THIS^.AssertEquals_BOOL(
	Expected 	:= assertionIsWrong,
	Actual 		:= THIS^.assertorContainer.wasAssertionWrong,
	Message 	:= messageStringBuilder.sOut
);
END_METHOD

(*

short summary
==================
This test method tests ``assert.times.long.valueIsEqualTo``
method of CNM_AssertionInterfaces library, 
it provides the possibility to handover test data via parameter 


.. <legal notes>

legal notes
=================
| SPDX-FileCopyrightText: © 2022 ekvip automation GmbH <info@ekvip.de>
| SPDX-License-Identifier: Apache-2.0
| For details check: Apache-2.0_

.. _Apache-2.0: https://www.apache.org/licenses/LICENSE-2.0

.. </legal notes>

parameters
==========

*)

METHOD testValueIsEqualTo 
VAR_INPUT
	(* for the test it's the parameter ``currentValue`` *)
	valueToTest	:LTIME;
	(* for the test it's the parameter ``expectedValue`` *)
	expected	:LTIME;
END_VAR
VAR
	(* just the expectation if the assertion to test must be worng or true *)
	assertionIsWrong		:BOOL;
	(* contains the format string for the test message *)
	message					:Tc2_System.T_MaxString;
	(* TwinCAT printf with the test message *)
	messageStringBuilder	:Tc2_Utilities.FB_FormatString;
	(* LTIME value of ``currentValue`` as string *)
	currentValueAsString	:STRING(22);
	(* LTIME value of ``expectedValue`` as string *)
	expectedValueAsString	:STRING(22);
END_VAR
THIS^.assertorContainer.resetAssertor();

assertionIsWrong := (valueToTest <> expected);

message := SEL(
	assertionIsWrong,
	'currentValue is %s expectedValue is %s assertion must be TRUE', 
	'currentValue is %s expectedValue is %s assertion must be FALSE'
);
currentValueAsString := TO_STRING(valueToTest);
expectedValueAsString := TO_STRING(expected);

messageStringBuilder(
	sFormat := message,
	arg1 := THIS^.AnyToArg(currentValueAsString),
	arg2 := THIS^.AnyToArg(expectedValueAsString)
);

THIS^.assertorContainer.assertor.assert.times.long.valueIsEqualTo(
	currentValue	:= valueToTest,
	expectedValue	:= expected,
	message			:= ''
);

THIS^.AssertEquals_BOOL(
	Expected 	:= assertionIsWrong,
	Actual 		:= THIS^.assertorContainer.wasAssertionWrong,
	Message 	:= messageStringBuilder.sOut
);
END_METHOD

(*

short summary
==================
This test method tests ``assert.times.long.valueIsGreaterThan``
method of CNM_AssertionInterfaces library, 
it provides the possibility to handover test data via parameter 


.. <legal notes>

legal notes
=================
| SPDX-FileCopyrightText: © 2022 ekvip automation GmbH <info@ekvip.de>
| SPDX-License-Identifier: Apache-2.0
| For details check: Apache-2.0_

.. _Apache-2.0: https://www.apache.org/licenses/LICENSE-2.0

.. </legal notes>

parameters
==========

*)

METHOD testValueIsGreaterThan 
VAR_INPUT
	(* for the test it's the parameter ``currentValue`` *)
	valueToTest	:LTIME;
	(* for the test it's the parameter ``lessValue`` *)
	lessValue	:LTIME;
END_VAR
VAR
	(* just the expectation if the assertion to test must be worng or true *)
	assertionIsWrong		:BOOL;
	(* contains the format string for the test message *)
	message					:Tc2_System.T_MaxString;
	(* TwinCAT printf with the test message *)
	messageStringBuilder	:Tc2_Utilities.FB_FormatString;
	(* LTIME value of ``currentValue`` as string *)
	currentValueAsString	:STRING(22);
	(* LTIME value of ``lessValue`` as string *)
	lessValueAsString		:STRING(22);
END_VAR
THIS^.assertorContainer.resetAssertor();

assertionIsWrong := (valueToTest <= lessValue);

message := SEL(
	assertionIsWrong,
	'currentValue is %s lessValue is %s assertion must be TRUE', 
	'currentValue is %s lessValue is %s assertion must be FALSE'
);
currentValueAsString := TO_STRING(valueToTest);
lessValueAsString := TO_STRING(lessValue);

messageStringBuilder(
	sFormat := message,
	arg1 := THIS^.AnyToArg(currentValueAsString),
	arg2 := THIS^.AnyToArg(lessValueAsString)
);

THIS^.assertorContainer.assertor.assert.times.long.valueIsGreaterThan(
	currentValue	:= valueToTest,
	lessValue		:= lessValue,
	message			:= ''
);

THIS^.AssertEquals_BOOL(
	Expected 	:= assertionIsWrong,
	Actual 		:= THIS^.assertorContainer.wasAssertionWrong,
	Message 	:= messageStringBuilder.sOut
);
END_METHOD

(*

short summary
==================
This test method tests ``assert.times.long.valueIsInRangeOf``
method of CNM_AssertionInterfaces library, 
it provides the possibility to handover test data via parameter 


.. <legal notes>

legal notes
=================
| SPDX-FileCopyrightText: © 2022 ekvip automation GmbH <info@ekvip.de>
| SPDX-License-Identifier: Apache-2.0
| For details check: Apache-2.0_

.. _Apache-2.0: https://www.apache.org/licenses/LICENSE-2.0

.. </legal notes>

parameters
==========

*)

METHOD testValueIsInRangeOf 
VAR_INPUT
	(* for the test it's the parameter ``lowerLimit`` *)
	lowerLimit	:LTIME;
	(* for the test it's the parameter ``currentValue`` *)
	valueToTest	:LTIME;
	(* for the test it's the parameter ``upperLimit`` *)
	upperLimit	:LTIME;
END_VAR
VAR
	(* just the expectation if the assertion to test must be worng or true *)
	assertionIsWrong		:BOOL;
	(* contains the format string for the test message *)
	message					:Tc2_System.T_MaxString;
	(* TwinCAT printf with the test message *)
	messageStringBuilder	:Tc2_Utilities.FB_FormatString;
	(* LTIME value of ``lowerLimit`` as string *)
	lowerLimitAsString		:STRING(22);
	(* LTIME value of ``currentValue`` as string *)
	currentValueAsString	:STRING(22);
	(* LTIME value of ``upperLimit`` as string *)
	upperLimitAsString		:STRING(22);

END_VAR
THIS^.assertorContainer.resetAssertor();

assertionIsWrong := ((
		valueToTest < lowerLimit
	) OR (
		valueToTest > upperLimit
	)
);

message := SEL(
	assertionIsWrong,
	'lowerLimit is %s currentValue is %s upperLimit is %s assertion must be TRUE', 
	'lowerLimit is %s currentValue is %s upperLimit is %s assertion must be FALSE'
);
lowerLimitAsString		:= TO_STRING(lowerLimit);
currentValueAsString	:= TO_STRING(valueToTest);
upperLimitAsString		:= TO_STRING(upperLimit);

messageStringBuilder(
	sFormat := message,
	arg1 := THIS^.AnyToArg(lowerLimitAsString),
	arg2 := THIS^.AnyToArg(currentValueAsString),
	arg3 := THIS^.AnyToArg(upperLimitAsString)
);

THIS^.assertorContainer.assertor.assert.times.long.valueIsInRangeOf(
	lowerLimit		:= lowerLimit,
	currentValue	:= valueToTest,
	upperLimit		:= upperLimit,
	message			:= ''
);

THIS^.AssertEquals_BOOL(
	Expected 	:= assertionIsWrong,
	Actual 		:= THIS^.assertorContainer.wasAssertionWrong,
	Message 	:= messageStringBuilder.sOut
);
END_METHOD

(*

short summary
==================
This test method tests ``assert.times.long.valueIsLessThan``
method of CNM_AssertionInterfaces library, 
it provides the possibility to handover test data via parameter 


.. <legal notes>

legal notes
=================
| SPDX-FileCopyrightText: © 2022 ekvip automation GmbH <info@ekvip.de>
| SPDX-License-Identifier: Apache-2.0
| For details check: Apache-2.0_

.. _Apache-2.0: https://www.apache.org/licenses/LICENSE-2.0

.. </legal notes>

parameters
==========

*)

METHOD testValueIsLessThan 
VAR_INPUT
	(* for the test it's the parameter ``currentValue`` *)
	valueToTest		:LTIME;
	(* for the test it's the parameter ``greaterValue`` *)
	greaterValue	:LTIME;
END_VAR
VAR
	(* just the expectation if the assertion to test must be worng or true *)
	assertionIsWrong		:BOOL;
	(* contains the format string for the test message *)
	message					:Tc2_System.T_MaxString;
	(* TwinCAT printf with the test message *)
	messageStringBuilder	:Tc2_Utilities.FB_FormatString;
	(* LTIME value of ``currentValue`` as string *)
	currentValueAsString	:STRING(22);
	(* LTIME value of ``greaterValue`` as string *)
	greaterValueAsString	:STRING(22);
END_VAR
THIS^.assertorContainer.resetAssertor();

assertionIsWrong := (valueToTest >= greaterValue);

message := SEL(
	assertionIsWrong,
	'currentValue is %s greaterValue is %s assertion must be TRUE', 
	'currentValue is %s greaterValue is %s assertion must be FALSE'
);
currentValueAsString := TO_STRING(valueToTest);
greaterValueAsString := TO_STRING(greaterValue);

messageStringBuilder(
	sFormat := message,
	arg1 := THIS^.AnyToArg(currentValueAsString),
	arg2 := THIS^.AnyToArg(greaterValueAsString)
);

THIS^.assertorContainer.assertor.assert.times.long.valueIsLessThan(
	currentValue	:= valueToTest,
	greaterValue	:= greaterValue,
	message			:= ''
);

THIS^.AssertEquals_BOOL(
	Expected 	:= assertionIsWrong,
	Actual 		:= THIS^.assertorContainer.wasAssertionWrong,
	Message 	:= messageStringBuilder.sOut
);
END_METHOD

(*

short summary
==================
This test method tests ``assert.times.long.valueIsMax``
method of CNM_AssertionInterfaces library, 
it provides the possibility to handover test data via parameter 


.. <legal notes>

legal notes
=================
| SPDX-FileCopyrightText: © 2022 ekvip automation GmbH <info@ekvip.de>
| SPDX-License-Identifier: Apache-2.0
| For details check: Apache-2.0_

.. _Apache-2.0: https://www.apache.org/licenses/LICENSE-2.0

.. </legal notes>

parameters
==========

*)

METHOD testValueIsMax 
VAR_INPUT
	(* for the test it's the parameter ``currentValue`` *)
	valueToTest		:LTIME;
	(* for the test it's the parameter ``greaterValue`` *)
	maximumValue	:LTIME;
END_VAR
VAR
	(* just the expectation if the assertion to test must be worng or true *)
	assertionIsWrong		:BOOL;
	(* contains the format string for the test message *)
	message					:Tc2_System.T_MaxString;
	(* TwinCAT printf with the test message *)
	messageStringBuilder	:Tc2_Utilities.FB_FormatString;
	(* LTIME value of ``currentValue`` as string *)
	currentValueAsString	:STRING(22);
	(* LTIME value of ``maximumValue`` as string *)
	maximumValueAsString	:STRING(22);
END_VAR
THIS^.assertorContainer.resetAssertor();

assertionIsWrong := (valueToTest > maximumValue);

message := SEL(
	assertionIsWrong,
	'currentValue is %s maximumValue is %s assertion must be TRUE', 
	'currentValue is %s maximumValue is %s assertion must be FALSE'
);
currentValueAsString := TO_STRING(valueToTest);
maximumValueAsString := TO_STRING(maximumValue);

messageStringBuilder(
	sFormat := message,
	arg1 := THIS^.AnyToArg(currentValueAsString),
	arg2 := THIS^.AnyToArg(maximumValueAsString)
);

THIS^.assertorContainer.assertor.assert.times.long.valueIsMax(
	currentValue	:= valueToTest,
	maximumValue	:= maximumValue,
	message			:= ''
);

THIS^.AssertEquals_BOOL(
	Expected 	:= assertionIsWrong,
	Actual 		:= THIS^.assertorContainer.wasAssertionWrong,
	Message 	:= messageStringBuilder.sOut
);
END_METHOD

(*

short summary
==================
This test method tests ``assert.times.long.valueIsMin``
method of CNM_AssertionInterfaces library, 
it provides the possibility to handover test data via parameter 


.. <legal notes>

legal notes
=================
| SPDX-FileCopyrightText: © 2022 ekvip automation GmbH <info@ekvip.de>
| SPDX-License-Identifier: Apache-2.0
| For details check: Apache-2.0_

.. _Apache-2.0: https://www.apache.org/licenses/LICENSE-2.0

.. </legal notes>

parameters
==========

*)

METHOD testValueIsMin 
VAR_INPUT
	(* for the test it's the parameter ``currentValue`` *)
	valueToTest		:LTIME;
	(* for the test it's the parameter ``greaterValue`` *)
	minimumValue	:LTIME;
END_VAR
VAR
	(* just the expectation if the assertion to test must be worng or true *)
	assertionIsWrong		:BOOL;
	(* contains the format string for the test message *)
	message					:Tc2_System.T_MaxString;
	(* TwinCAT printf with the test message *)
	messageStringBuilder	:Tc2_Utilities.FB_FormatString;
	(* LTIME value of ``currentValue`` as string *)
	currentValueAsString	:STRING(22);
	(* LTIME value of ``minimumValue`` as string *)
	minimumValueAsString	:STRING(22);
END_VAR
THIS^.assertorContainer.resetAssertor();

assertionIsWrong := (valueToTest < minimumValue);

message := SEL(
	assertionIsWrong,
	'currentValue is %s minimumValue is %s assertion must be TRUE', 
	'currentValue is %s minimumValue is %s assertion must be FALSE'
);
currentValueAsString := TO_STRING(valueToTest);
minimumValueAsString := TO_STRING(minimumValue);

messageStringBuilder(
	sFormat := message,
	arg1 := THIS^.AnyToArg(currentValueAsString),
	arg2 := THIS^.AnyToArg(minimumValueAsString)
);

THIS^.assertorContainer.assertor.assert.times.long.valueIsMin(
	currentValue	:= valueToTest,
	minimumValue	:= minimumValue,
	message			:= ''
);

THIS^.AssertEquals_BOOL(
	Expected 	:= assertionIsWrong,
	Actual 		:= THIS^.assertorContainer.wasAssertionWrong,
	Message 	:= messageStringBuilder.sOut
);
END_METHOD

(*

short summary
==================
This test method tests ``assert.times.long.valueIsNotEqualTo``
method of CNM_AssertionInterfaces library, 
it provides the possibility to handover test data via parameter 


.. <legal notes>

legal notes
=================
| SPDX-FileCopyrightText: © 2022 ekvip automation GmbH <info@ekvip.de>
| SPDX-License-Identifier: Apache-2.0
| For details check: Apache-2.0_

.. _Apache-2.0: https://www.apache.org/licenses/LICENSE-2.0

.. </legal notes>

parameters
==========

*)

METHOD testValueIsNotEqualTo 
VAR_INPUT
	(* for the test it's the parameter ``currentValue`` *)
	valueToTest		:LTIME;
	(* for the test it's the parameter ``unexpectedValue`` *)
	unexpectedValue	:LTIME;
END_VAR
VAR
	(* just the expectation if the assertion to test must be worng or true *)
	assertionIsWrong		:BOOL;
	(* contains the format string for the test message *)
	message					:Tc2_System.T_MaxString;
	(* TwinCAT printf with the test message *)
	messageStringBuilder	:Tc2_Utilities.FB_FormatString;
	(* LTIME value of ``currentValue`` as string *)
	currentValueAsString	:STRING(22);
	(* LTIME value of ``unexpectedValue`` as string *)
	unexpectedValueAsString	:STRING(22);
END_VAR
THIS^.assertorContainer.resetAssertor();

assertionIsWrong := (valueToTest = unexpectedValue);

message := SEL(
	assertionIsWrong,
	'currentValue is %s expectedValue is %s assertion must be TRUE', 
	'currentValue is %s expectedValue is %s assertion must be FALSE'
);
currentValueAsString := TO_STRING(valueToTest);
unexpectedValueAsString := TO_STRING(unexpectedValue);

messageStringBuilder(
	sFormat := message,
	arg1 := THIS^.AnyToArg(currentValueAsString),
	arg2 := THIS^.AnyToArg(unexpectedValueAsString)
);

THIS^.assertorContainer.assertor.assert.times.long.valueIsNotEqualTo(
	currentValue	:= valueToTest,
	unexpectedValue	:= unexpectedValue,
	message			:= ''
);

THIS^.AssertEquals_BOOL(
	Expected 	:= assertionIsWrong,
	Actual 		:= THIS^.assertorContainer.wasAssertionWrong,
	Message 	:= messageStringBuilder.sOut
);
END_METHOD

END_FUNCTION_BLOCK

// ---- AssertionTester/AssertionTests/TimeAssertions/classes/TimeAssertionsTests.TcPOU
(*

short summary
==================
This class tests all methods of TIME assertions
with various combinations of inputs and checks expected 
outputs are satisfied or not

.. <legal notes>

legal notes
=================
| SPDX-FileCopyrightText: © 2022 ekvip automation GmbH <info@ekvip.de>
| SPDX-License-Identifier: Apache-2.0
| For details check: Apache-2.0_

.. _Apache-2.0: https://www.apache.org/licenses/LICENSE-2.0

.. </legal notes>

methods and properties
======================

*)


FUNCTION_BLOCK TimeAssertionsTests EXTENDS AbstractAssertorTest
VAR
	
END_VAR
VAR CONSTANT
	(* prefix to unify the test names *)
	TEST_NAME_PREFIX		:STRING := 'assert.times.simple.';
	(* max value of a DWORD *)
	{attribute 'hide'}
	MAX_DWORD				:DWORD := 16#FFFF_FFFF;
	(* min value of a DWORD *)
	{attribute 'hide'}
	MIN_DWORD				:DWORD := 16#0000_0000;
	(* only the msb is set *)
	{attribute 'hide'}
	MSB_ONLY				:DWORD := 16#8000_0000;
	(* only the msb is set *)
	{attribute 'hide'}
	LSB_ONLY				:DWORD := 16#0000_0001;
	(* all bits set except the msb *)
	{attribute 'hide'}
	WITHOUT_MSB 			:DWORD := 16#7FFF_FFFF;
	(* for every nibble is the msb set only *)
	{attribute 'hide'}
	ALL_NIBBLE_MSB			:DWORD := 16#8888_8888;
	(* for every nibble is the msb unset only *)
	{attribute 'hide'}
	WITHOUT_NIBBLE_MSB		:DWORD := 16#7777_7777;
	(* for every nibble is the lsb set only *)
	{attribute 'hide'}
	ALL_NIBBLE_LSB			:DWORD := 16#1111_1111;
	(* every bit is set except the lsb *)
	{attribute 'hide'}
	LSB_IS_UNSET			:DWORD := 16#FFFF_FFFE;
	(* max vale of time *)
	TIME_MAX				:TIME := TO_TIME(MAX_DWORD);
	(* min vale of time *)
	TIME_MIN				:TIME := TO_TIME(MIN_DWORD);
	(* only the msb is set *)
	TIME_MSB_ONLY			:TIME := TO_TIME(MSB_ONLY);
	(* all bits set except the msb *)
	TIME_WITHOUT_MSB 		:TIME := TO_TIME(WITHOUT_MSB);
	(* for every nibble is the msb set only *)
	TIME_ALL_NIBBLE_MSB		:TIME := TO_TIME(ALL_NIBBLE_MSB);
	(* for every nibble is the msb unset only *)
	TIME_WITHOUT_NIBBLE_MSB	:TIME := TO_TIME(WITHOUT_NIBBLE_MSB);
	(* for every nibble is the lsb set only *)
	TIME_ALL_NIBBLE_LSB		:TIME := TO_TIME(ALL_NIBBLE_LSB);	
	(* every bit is set except the lsb *)
	TIME_LSB_IS_UNSET		:TIME := TO_TIME(LSB_IS_UNSET);
	(* only the msb is set *)
	TIME_LSB_ONLY			:TIME := TO_TIME(LSB_ONLY);
END_VAR

THIS^.runTimeHasExpired();
THIS^.runTimeHasNotExpired();
THIS^.runValueIsEqualToTests();
THIS^.runValueIsGreaterThanTests();
THIS^.runValueIsInRangeOfTests();
THIS^.runValueIsLessThanTests();
THIS^.runValueIsMaxTests();
THIS^.runValueIsMinTests();
THIS^.runValueIsNotEqualToTests();

(*

short summary
==================
This test method is a helper function to create a unified test name

.. <legal notes>

legal notes
=================
| SPDX-FileCopyrightText: © 2022 ekvip automation GmbH <info@ekvip.de>
| SPDX-License-Identifier: Apache-2.0
| For details check: Apache-2.0_

.. _Apache-2.0: https://www.apache.org/licenses/LICENSE-2.0

.. </legal notes>

parameters
==========

*)

METHOD PROTECTED getTestNameFor :Tc2_System.T_MaxString
VAR_INPUT
	(* name of the method to test, to create a unified test name *)
	nameOfMethodToTest	:Tc2_System.T_MaxString;
END_VAR
getTestNameFor := Tc2_Standard.CONCAT(THIS^.TEST_NAME_PREFIX, nameOfMethodToTest);
END_METHOD

(*

short summary
=================
This method returns the passed time since the timestamp was created
(helper method of CNM_AssertionInterfaces)

.. <legal notes>

legal notes
=================
| SPDX-FileCopyrightText: © 2022 ekvip automation GmbH <info@ekvip.de>
| SPDX-License-Identifier: Apache-2.0
| For details check: Apache-2.0_

.. _Apache-2.0: https://www.apache.org/licenses/LICENSE-2.0

.. </legal notes>

parameters
=================
:return: passed time since ``startTime``

*)

METHOD PROTECTED getTimePassed :TIME
VAR_INPUT
	(* timestamp start *)
	startTime	:TIME;
END_VAR
VAR
	(* current time to calculate the passed time *)
	currentTime	:TIME;
END_VAR
currentTime := TIME();
IF (currentTime > startTime) THEN
	getTimePassed := (currentTime - startTime);
ELSE
	getTimePassed := ((THIS^.TIME_MAX - startTime) + currentTime);
END_IF
END_METHOD

(*

short summary
==================
This test method tests ``assert.times.simple.timeHasExpired``
method of CNM_AssertionInterfaces library with various inputs

.. <legal notes>

legal notes
=================
| SPDX-FileCopyrightText: © 2022 ekvip automation GmbH <info@ekvip.de>
| SPDX-License-Identifier: Apache-2.0
| For details check: Apache-2.0_

.. _Apache-2.0: https://www.apache.org/licenses/LICENSE-2.0

.. </legal notes>

*)

METHOD runTimeHasExpired
RETURN (NOT TcUnit.TEST_ORDERED(THIS^.getTestNameFor('timeHasExpired')));

THIS^.testTimeHasExpired(
	valueToTest := THIS^.TIME_MAX,
	expiring := THIS^.TIME_MAX
);
THIS^.testTimeHasExpired(
	valueToTest := THIS^.TIME_MIN,
	expiring := THIS^.TIME_MIN
);
THIS^.testTimeHasExpired(
	valueToTest := THIS^.TIME_MAX,
	expiring := THIS^.TIME_MIN
);
THIS^.testTimeHasExpired(
	valueToTest := THIS^.TIME_MIN,
	expiring := THIS^.TIME_MAX
);
THIS^.testTimeHasExpired(
	valueToTest := THIS^.TIME_ALL_NIBBLE_LSB,
	expiring := THIS^.TIME_ALL_NIBBLE_LSB
);	
THIS^.testTimeHasExpired(
	valueToTest := THIS^.TIME_ALL_NIBBLE_LSB,
	expiring := THIS^.TIME_ALL_NIBBLE_MSB
);
THIS^.testTimeHasExpired(
	valueToTest := THIS^.TIME_ALL_NIBBLE_MSB,
	expiring := THIS^.TIME_ALL_NIBBLE_LSB
);
THIS^.testTimeHasExpired(
	valueToTest := THIS^.TIME_LSB_ONLY,
	expiring := THIS^.TIME_MSB_ONLY
);
THIS^.testTimeHasExpired(
	valueToTest := THIS^.TIME_MSB_ONLY,
	expiring := THIS^.TIME_MSB_ONLY
);
THIS^.testTimeHasExpired(
	valueToTest := THIS^.TIME_MSB_ONLY,
	expiring := THIS^.TIME_LSB_ONLY
);
THIS^.testTimeHasExpired(
	valueToTest := THIS^.TIME_LSB_IS_UNSET,
	expiring := THIS^.TIME_MAX
);
THIS^.testTimeHasExpired(
	valueToTest := THIS^.TIME_MAX,
	expiring := THIS^.TIME_LSB_IS_UNSET
);

TcUnit.TEST_FINISHED();
END_METHOD

(*

short summary
==================
This test method tests ``assert.times.simple.timeHasNotExpired``
method of CNM_AssertionInterfaces library with various inputs

.. <legal notes>

legal notes
=================
| SPDX-FileCopyrightText: © 2022 ekvip automation GmbH <info@ekvip.de>
| SPDX-License-Identifier: Apache-2.0
| For details check: Apache-2.0_

.. _Apache-2.0: https://www.apache.org/licenses/LICENSE-2.0

.. </legal notes>

*)

METHOD runTimeHasNotExpired
RETURN (NOT TcUnit.TEST_ORDERED(THIS^.getTestNameFor('timeHasNotExpired')));

THIS^.testTimeHasExpired(
	valueToTest := THIS^.TIME_MAX,
	expiring := THIS^.TIME_MAX
);
THIS^.testTimeHasExpired(
	valueToTest := THIS^.TIME_MIN,
	expiring := THIS^.TIME_MIN
);
THIS^.testTimeHasExpired(
	valueToTest := THIS^.TIME_MAX,
	expiring := THIS^.TIME_MIN
);
THIS^.testTimeHasExpired(
	valueToTest := THIS^.TIME_MIN,
	expiring := THIS^.TIME_MAX
);
THIS^.testTimeHasExpired(
	valueToTest := THIS^.TIME_ALL_NIBBLE_LSB,
	expiring := THIS^.TIME_ALL_NIBBLE_LSB
);	
THIS^.testTimeHasExpired(
	valueToTest := THIS^.TIME_ALL_NIBBLE_LSB,
	expiring := THIS^.TIME_ALL_NIBBLE_MSB
);
THIS^.testTimeHasExpired(
	valueToTest := THIS^.TIME_ALL_NIBBLE_MSB,
	expiring := THIS^.TIME_ALL_NIBBLE_LSB
);
THIS^.testTimeHasExpired(
	valueToTest := THIS^.TIME_LSB_ONLY,
	expiring := THIS^.TIME_MSB_ONLY
);
THIS^.testTimeHasExpired(
	valueToTest := THIS^.TIME_MSB_ONLY,
	expiring := THIS^.TIME_MSB_ONLY
);
THIS^.testTimeHasExpired(
	valueToTest := THIS^.TIME_MSB_ONLY,
	expiring := THIS^.TIME_LSB_ONLY
);
THIS^.testTimeHasExpired(
	valueToTest := THIS^.TIME_LSB_IS_UNSET,
	expiring := THIS^.TIME_MAX
);
THIS^.testTimeHasExpired(
	valueToTest := THIS^.TIME_MAX,
	expiring := THIS^.TIME_LSB_IS_UNSET
);

TcUnit.TEST_FINISHED();
END_METHOD

(*

short summary
==================
This test method tests ``assert.times.simple.valueIsEqualTo``
method of CNM_AssertionInterfaces library with various inputs

.. <legal notes>

legal notes
=================
| SPDX-FileCopyrightText: © 2022 ekvip automation GmbH <info@ekvip.de>
| SPDX-License-Identifier: Apache-2.0
| For details check: Apache-2.0_

.. _Apache-2.0: https://www.apache.org/licenses/LICENSE-2.0

.. </legal notes>

*)

METHOD runValueIsEqualToTests
RETURN (NOT TcUnit.TEST_ORDERED(THIS^.getTestNameFor('valueIsEqualTo')));

THIS^.testValueIsEqualTo(
	valueToTest := THIS^.TIME_MAX,
	expected := THIS^.TIME_MAX
);
THIS^.testValueIsEqualTo(
	valueToTest := THIS^.TIME_MIN,
	expected := THIS^.TIME_MIN
);
THIS^.testValueIsEqualTo(
	valueToTest := THIS^.TIME_MIN,
	expected := THIS^.TIME_MAX
);
THIS^.testValueIsEqualTo(
	valueToTest := THIS^.TIME_MAX,
	expected := THIS^.TIME_MIN
);
THIS^.testValueIsEqualTo(
	valueToTest := THIS^.TIME_ALL_NIBBLE_LSB,
	expected := THIS^.TIME_ALL_NIBBLE_LSB
);
THIS^.testValueIsEqualTo(
	valueToTest := THIS^.TIME_LSB_ONLY,
	expected := THIS^.TIME_MSB_ONLY
);
THIS^.testValueIsEqualTo(
	valueToTest := THIS^.TIME_MSB_ONLY,
	expected := THIS^.TIME_MSB_ONLY
);
THIS^.testValueIsEqualTo(
	valueToTest := THIS^.TIME_MSB_ONLY,
	expected := THIS^.TIME_LSB_ONLY
);

TcUnit.TEST_FINISHED();
END_METHOD

(*

short summary
==================
This test method tests ``assert.times.simple.valueIsGreaterThan``
method of CNM_AssertionInterfaces library with various inputs

.. <legal notes>

legal notes
=================
| SPDX-FileCopyrightText: © 2022 ekvip automation GmbH <info@ekvip.de>
| SPDX-License-Identifier: Apache-2.0
| For details check: Apache-2.0_

.. _Apache-2.0: https://www.apache.org/licenses/LICENSE-2.0

.. </legal notes>

*)

METHOD runValueIsGreaterThanTests
RETURN (NOT TcUnit.TEST_ORDERED(THIS^.getTestNameFor('valueIsGreaterThan')));

THIS^.testValueIsGreaterThan(
	valueToTest := THIS^.TIME_MAX,
	lessValue := THIS^.TIME_MAX
);
THIS^.testValueIsGreaterThan(
	valueToTest := THIS^.TIME_MIN,
	lessValue := THIS^.TIME_MIN
);
THIS^.testValueIsGreaterThan(
	valueToTest := THIS^.TIME_MIN,
	lessValue := THIS^.TIME_MAX
);
THIS^.testValueIsGreaterThan(
	valueToTest := THIS^.TIME_MAX,
	lessValue := THIS^.TIME_MIN
);
THIS^.testValueIsGreaterThan(
	valueToTest := THIS^.TIME_ALL_NIBBLE_LSB,
	lessValue := THIS^.TIME_ALL_NIBBLE_LSB
);
THIS^.testValueIsGreaterThan(
	valueToTest := THIS^.TIME_ALL_NIBBLE_MSB,
	lessValue := THIS^.TIME_ALL_NIBBLE_LSB
);
THIS^.testValueIsGreaterThan(
	valueToTest := THIS^.TIME_ALL_NIBBLE_LSB,
	lessValue := THIS^.TIME_ALL_NIBBLE_MSB
);
THIS^.testValueIsGreaterThan(
	valueToTest := THIS^.TIME_LSB_ONLY,
	lessValue := THIS^.TIME_MSB_ONLY
);
THIS^.testValueIsGreaterThan(
	valueToTest := THIS^.TIME_MSB_ONLY,
	lessValue := THIS^.TIME_MSB_ONLY
);
THIS^.testValueIsGreaterThan(
	valueToTest := THIS^.TIME_MSB_ONLY,
	lessValue := THIS^.TIME_LSB_ONLY
);
THIS^.testValueIsGreaterThan(
	valueToTest := THIS^.TIME_LSB_IS_UNSET,
	lessValue := THIS^.TIME_MAX
);
THIS^.testValueIsGreaterThan(
	valueToTest := THIS^.TIME_MAX,
	lessValue := THIS^.TIME_LSB_IS_UNSET
);

TcUnit.TEST_FINISHED();
END_METHOD

(*

short summary
==================
This test method tests ``assert.times.simple.valueIsInRangeOf``
method of CNM_AssertionInterfaces library with various inputs

.. <legal notes>

legal notes
=================
| SPDX-FileCopyrightText: © 2022 ekvip automation GmbH <info@ekvip.de>
| SPDX-License-Identifier: Apache-2.0
| For details check: Apache-2.0_

.. _Apache-2.0: https://www.apache.org/licenses/LICENSE-2.0

.. </legal notes>

*)

METHOD runValueIsInRangeOfTests
RETURN (NOT TcUnit.TEST_ORDERED(THIS^.getTestNameFor('valueIsInRangeOf')));

THIS^.testValueIsInRangeOf(
	lowerLimit := THIS^.TIME_MIN,
	valueToTest := THIS^.TIME_MAX,
	upperLimit	:= THIS^.TIME_MAX
);
THIS^.testValueIsInRangeOf(
	lowerLimit := THIS^.TIME_MIN,
	valueToTest := THIS^.TIME_MIN,
	upperLimit	:= THIS^.TIME_MAX
);
THIS^.testValueIsInRangeOf(
	lowerLimit := THIS^.TIME_MAX,
	valueToTest := THIS^.TIME_MAX,
	upperLimit	:= THIS^.TIME_MIN
);
THIS^.testValueIsInRangeOf(
	lowerLimit := THIS^.TIME_MAX,
	valueToTest := THIS^.TIME_MIN,
	upperLimit	:= THIS^.TIME_MIN
);
THIS^.testValueIsInRangeOf(
	lowerLimit := THIS^.TIME_LSB_IS_UNSET,
	valueToTest := THIS^.TIME_MIN,
	upperLimit	:= THIS^.TIME_MAX
);
THIS^.testValueIsInRangeOf(
	lowerLimit := THIS^.TIME_MIN,
	valueToTest := THIS^.TIME_LSB_IS_UNSET,
	upperLimit	:= THIS^.TIME_MAX
);
THIS^.testValueIsInRangeOf(
	lowerLimit := THIS^.TIME_LSB_IS_UNSET,
	valueToTest := THIS^.TIME_LSB_IS_UNSET,
	upperLimit	:= THIS^.TIME_LSB_IS_UNSET
);
THIS^.testValueIsInRangeOf(
	lowerLimit := THIS^.TIME_ALL_NIBBLE_LSB,
	valueToTest := THIS^.TIME_LSB_IS_UNSET,
	upperLimit	:= THIS^.TIME_ALL_NIBBLE_MSB
);
THIS^.testValueIsInRangeOf(
	lowerLimit := THIS^.TIME_LSB_IS_UNSET,
	valueToTest := THIS^.TIME_ALL_NIBBLE_LSB,
	upperLimit	:= THIS^.TIME_ALL_NIBBLE_MSB
);
THIS^.testValueIsInRangeOf(
	lowerLimit := THIS^.TIME_LSB_ONLY,
	valueToTest := THIS^.TIME_WITHOUT_MSB,
	upperLimit	:= THIS^.TIME_MSB_ONLY
);
THIS^.testValueIsInRangeOf(
	lowerLimit := THIS^.TIME_WITHOUT_MSB,
	valueToTest := THIS^.TIME_LSB_ONLY,
	upperLimit	:= THIS^.TIME_MSB_ONLY
);
THIS^.testValueIsInRangeOf(
	lowerLimit := THIS^.TIME_WITHOUT_NIBBLE_MSB,
	valueToTest := THIS^.TIME_MAX,
	upperLimit	:= THIS^.TIME_ALL_NIBBLE_MSB
);
THIS^.testValueIsInRangeOf(
	lowerLimit := THIS^.TIME_WITHOUT_NIBBLE_MSB,
	valueToTest := THIS^.TIME_MIN,
	upperLimit	:= THIS^.TIME_ALL_NIBBLE_MSB
);
THIS^.testValueIsInRangeOf(
	lowerLimit := THIS^.TIME_WITHOUT_NIBBLE_MSB,
	valueToTest := THIS^.TIME_WITHOUT_NIBBLE_MSB,
	upperLimit	:= THIS^.TIME_ALL_NIBBLE_MSB
);
THIS^.testValueIsInRangeOf(
	lowerLimit := THIS^.TIME_WITHOUT_NIBBLE_MSB,
	valueToTest := THIS^.TIME_ALL_NIBBLE_MSB,
	upperLimit	:= THIS^.TIME_ALL_NIBBLE_MSB
);

TcUnit.TEST_FINISHED();
END_METHOD

(*

short summary
==================
This test method tests ``assert.times.simple.valueIsLessThan``
method of CNM_AssertionInterfaces library with various inputs

.. <legal notes>

legal notes
=================
| SPDX-FileCopyrightText: © 2022 ekvip automation GmbH <info@ekvip.de>
| SPDX-License-Identifier: Apache-2.0
| For details check: Apache-2.0_

.. _Apache-2.0: https://www.apache.org/licenses/LICENSE-2.0

.. </legal notes>

*)

METHOD runValueIsLessThanTests
RETURN (NOT TcUnit.TEST_ORDERED(THIS^.getTestNameFor('valueIsLessThan')));

THIS^.testValueIsLessThan(
	valueToTest := THIS^.TIME_MAX,
	greaterValue := THIS^.TIME_MAX
);
THIS^.testValueIsLessThan(
	valueToTest := THIS^.TIME_MIN,
	greaterValue := THIS^.TIME_MIN
);
THIS^.testValueIsLessThan(
	valueToTest := THIS^.TIME_MIN,
	greaterValue := THIS^.TIME_MAX
);
THIS^.testValueIsLessThan(
	valueToTest := THIS^.TIME_MAX,
	greaterValue := THIS^.TIME_MIN
);
THIS^.testValueIsLessThan(
	valueToTest := THIS^.TIME_ALL_NIBBLE_LSB,
	greaterValue := THIS^.TIME_ALL_NIBBLE_LSB
);
THIS^.testValueIsLessThan(
	valueToTest := THIS^.TIME_ALL_NIBBLE_MSB,
	greaterValue := THIS^.TIME_ALL_NIBBLE_LSB
);
THIS^.testValueIsLessThan(
	valueToTest := THIS^.TIME_ALL_NIBBLE_LSB,
	greaterValue := THIS^.TIME_ALL_NIBBLE_MSB
);
THIS^.testValueIsLessThan(
	valueToTest := THIS^.TIME_LSB_ONLY,
	greaterValue := THIS^.TIME_MSB_ONLY
);
THIS^.testValueIsLessThan(
	valueToTest := THIS^.TIME_MSB_ONLY,
	greaterValue := THIS^.TIME_MSB_ONLY
);
THIS^.testValueIsLessThan(
	valueToTest := THIS^.TIME_MSB_ONLY,
	greaterValue := THIS^.TIME_LSB_ONLY
);
THIS^.testValueIsLessThan(
	valueToTest := THIS^.TIME_LSB_IS_UNSET,
	greaterValue := THIS^.TIME_MAX
);
THIS^.testValueIsLessThan(
	valueToTest := THIS^.TIME_MAX,
	greaterValue := THIS^.TIME_LSB_IS_UNSET
);

TcUnit.TEST_FINISHED();
END_METHOD

(*

short summary
==================
This test method tests ``assert.times.simple.valueIsMax``
method of CNM_AssertionInterfaces library with various inputs

.. <legal notes>

legal notes
=================
| SPDX-FileCopyrightText: © 2022 ekvip automation GmbH <info@ekvip.de>
| SPDX-License-Identifier: Apache-2.0
| For details check: Apache-2.0_

.. _Apache-2.0: https://www.apache.org/licenses/LICENSE-2.0

.. </legal notes>

*)

METHOD runValueIsMaxTests
RETURN (NOT TcUnit.TEST_ORDERED(THIS^.getTestNameFor('valueIsMax')));

THIS^.testValueIsMax(
	valueToTest := THIS^.TIME_MAX,
	maximumValue := THIS^.TIME_MAX
);
THIS^.testValueIsMax(
	valueToTest := THIS^.TIME_MIN,
	maximumValue := THIS^.TIME_MIN
);
THIS^.testValueIsMax(
	valueToTest := THIS^.TIME_MIN,
	maximumValue := THIS^.TIME_MAX
);
THIS^.testValueIsMax(
	valueToTest := THIS^.TIME_MAX,
	maximumValue := THIS^.TIME_MIN
);
THIS^.testValueIsMax(
	valueToTest := THIS^.TIME_ALL_NIBBLE_LSB,
	maximumValue := THIS^.TIME_ALL_NIBBLE_LSB
);
THIS^.testValueIsMax(
	valueToTest := THIS^.TIME_ALL_NIBBLE_MSB,
	maximumValue := THIS^.TIME_ALL_NIBBLE_LSB
);
THIS^.testValueIsMax(
	valueToTest := THIS^.TIME_ALL_NIBBLE_LSB,
	maximumValue := THIS^.TIME_ALL_NIBBLE_MSB
);
THIS^.testValueIsMax(
	valueToTest := THIS^.TIME_LSB_ONLY,
	maximumValue := THIS^.TIME_MSB_ONLY
);
THIS^.testValueIsMax(
	valueToTest := THIS^.TIME_MSB_ONLY,
	maximumValue := THIS^.TIME_MSB_ONLY
);
THIS^.testValueIsMax(
	valueToTest := THIS^.TIME_MSB_ONLY,
	maximumValue := THIS^.TIME_LSB_ONLY
);
THIS^.testValueIsMax(
	valueToTest := THIS^.TIME_LSB_IS_UNSET,
	maximumValue := THIS^.TIME_MAX
);
THIS^.testValueIsMax(
	valueToTest := THIS^.TIME_MAX,
	maximumValue := THIS^.TIME_LSB_IS_UNSET
);

TcUnit.TEST_FINISHED();
END_METHOD

(*

short summary
==================
This test method tests ``assert.times.simple.valueIsMin``
method of CNM_AssertionInterfaces library with various inputs

.. <legal notes>

legal notes
=================
| SPDX-FileCopyrightText: © 2022 ekvip automation GmbH <info@ekvip.de>
| SPDX-License-Identifier: Apache-2.0
| For details check: Apache-2.0_

.. _Apache-2.0: https://www.apache.org/licenses/LICENSE-2.0

.. </legal notes>

*)

METHOD runValueIsMinTests
RETURN (NOT TcUnit.TEST_ORDERED(THIS^.getTestNameFor('valueIsMin')));

THIS^.testValueIsMin(
	valueToTest := THIS^.TIME_MAX,
	minimumValue := THIS^.TIME_MAX
);
THIS^.testValueIsMin(
	valueToTest := THIS^.TIME_MIN,
	minimumValue := THIS^.TIME_MIN
);
THIS^.testValueIsMin(
	valueToTest := THIS^.TIME_MIN,
	minimumValue := THIS^.TIME_MAX
);
THIS^.testValueIsMin(
	valueToTest := THIS^.TIME_MAX,
	minimumValue := THIS^.TIME_MIN
);
THIS^.testValueIsMin(
	valueToTest := THIS^.TIME_ALL_NIBBLE_LSB,
	minimumValue := THIS^.TIME_ALL_NIBBLE_LSB
);
THIS^.testValueIsMin(
	valueToTest := THIS^.TIME_ALL_NIBBLE_MSB,
	minimumValue := THIS^.TIME_ALL_NIBBLE_LSB
);
THIS^.testValueIsMin(
	valueToTest := THIS^.TIME_ALL_NIBBLE_LSB,
	minimumValue := THIS^.TIME_ALL_NIBBLE_MSB
);
THIS^.testValueIsMin(
	valueToTest := THIS^.TIME_LSB_ONLY,
	minimumValue := THIS^.TIME_MSB_ONLY
);
THIS^.testValueIsMin(
	valueToTest := THIS^.TIME_MSB_ONLY,
	minimumValue := THIS^.TIME_MSB_ONLY
);
THIS^.testValueIsMin(
	valueToTest := THIS^.TIME_MSB_ONLY,
	minimumValue := THIS^.TIME_LSB_ONLY
);
THIS^.testValueIsMin(
	valueToTest := THIS^.TIME_LSB_IS_UNSET,
	minimumValue := THIS^.TIME_MAX
);
THIS^.testValueIsMin(
	valueToTest := THIS^.TIME_MAX,
	minimumValue := THIS^.TIME_LSB_IS_UNSET
);

TcUnit.TEST_FINISHED();
END_METHOD

(*

short summary
==================
This test method tests ``assert.times.simple.valueIsNotEqualTo``
method of CNM_AssertionInterfaces library with various inputs

.. <legal notes>

legal notes
=================
| SPDX-FileCopyrightText: © 2022 ekvip automation GmbH <info@ekvip.de>
| SPDX-License-Identifier: Apache-2.0
| For details check: Apache-2.0_

.. _Apache-2.0: https://www.apache.org/licenses/LICENSE-2.0

.. </legal notes>

*)

METHOD runValueIsNotEqualToTests
RETURN (NOT TcUnit.TEST_ORDERED(THIS^.getTestNameFor('valueIsNotEqualTo')));

THIS^.testValueIsNotEqualTo(
	valueToTest := THIS^.TIME_MAX,
	unexpectedValue := THIS^.TIME_MAX
);
THIS^.testValueIsNotEqualTo(
	valueToTest := THIS^.TIME_MIN,
	unexpectedValue := THIS^.TIME_MIN
);
THIS^.testValueIsNotEqualTo(
	valueToTest := THIS^.TIME_MIN,
	unexpectedValue := THIS^.TIME_MAX
);
THIS^.testValueIsNotEqualTo(
	valueToTest := THIS^.TIME_MAX,
	unexpectedValue := THIS^.TIME_MIN
);
THIS^.testValueIsNotEqualTo(
	valueToTest := THIS^.TIME_ALL_NIBBLE_LSB,
	unexpectedValue := THIS^.TIME_ALL_NIBBLE_LSB
);
THIS^.testValueIsNotEqualTo(
	valueToTest := THIS^.TIME_LSB_ONLY,
	unexpectedValue := THIS^.TIME_MSB_ONLY
);
THIS^.testValueIsNotEqualTo(
	valueToTest := THIS^.TIME_MSB_ONLY,
	unexpectedValue := THIS^.TIME_MSB_ONLY
);
THIS^.testValueIsNotEqualTo(
	valueToTest := THIS^.TIME_MSB_ONLY,
	unexpectedValue := THIS^.TIME_LSB_ONLY
);

TcUnit.TEST_FINISHED();
END_METHOD

(*

short summary
==================
This test method tests ``assert.times.simple.timeHasExpired``
method of CNM_AssertionInterfaces library, 
it provides the possibility to handover test data via parameter 


.. <legal notes>

legal notes
=================
| SPDX-FileCopyrightText: © 2022 ekvip automation GmbH <info@ekvip.de>
| SPDX-License-Identifier: Apache-2.0
| For details check: Apache-2.0_

.. _Apache-2.0: https://www.apache.org/licenses/LICENSE-2.0

.. </legal notes>

parameters
==========

*)


METHOD testTimeHasExpired 
VAR_INPUT
	(* for the test it's the parameter ``timestamp`` *)
	valueToTest	:TIME;
	(* for the test it's the parameter ``expiringTime`` *)
	expiring	:TIME;
END_VAR
VAR
	(* just the expectation if the assertion to test must be wrong or true *)
	assertionIsWrong		:BOOL;
	(* contains the format string for the test message *)
	message					:Tc2_System.T_MaxString;
	(* TwinCAT printf with the test message *)
	messageStringBuilder	:Tc2_Utilities.FB_FormatString;
	(* TIME value of ``expiringTime`` as string *)
	expiringTimeAsString	:STRING(22);
	(* TIME value of ``expectedValue`` as string *)
	timestampAsString		:STRING(22);
END_VAR
THIS^.assertorContainer.resetAssertor();

assertionIsWrong := (getTimePassed(startTime := valueToTest) < expiring);

message := SEL(
	assertionIsWrong,
	'timestamp is %s expiringTime is %s assertion must be TRUE', 
	'timestamp is %s expiringTime is %s assertion must be FALSE'
);
timestampAsString := TO_STRING(valueToTest);
expiringTimeAsString := TO_STRING(expiring);

messageStringBuilder(
	sFormat := message,
	arg1 := THIS^.AnyToArg(timestampAsString),
	arg2 := THIS^.AnyToArg(expiringTimeAsString)
);

THIS^.assertorContainer.assertor.assert.times.simple.timeHasExpired(
	timestamp		:= valueToTest,
	expiringTime	:= expiring,
	message			:= ''
);

THIS^.AssertEquals_BOOL(
	Expected 	:= assertionIsWrong,
	Actual 		:= THIS^.assertorContainer.wasAssertionWrong,
	Message 	:= messageStringBuilder.sOut
);
END_METHOD

(*

short summary
==================
This test method tests ``assert.times.simple.timeHasNotExpired``
method of CNM_AssertionInterfaces library, 
it provides the possibility to handover test data via parameter 


.. <legal notes>

legal notes
=================
| SPDX-FileCopyrightText: © 2022 ekvip automation GmbH <info@ekvip.de>
| SPDX-License-Identifier: Apache-2.0
| For details check: Apache-2.0_

.. _Apache-2.0: https://www.apache.org/licenses/LICENSE-2.0

.. </legal notes>

parameters
==========

*)


METHOD testTimeHasNotExpired 
VAR_INPUT
	(* for the test it's the parameter ``timestamp`` *)
	valueToTest	:TIME;
	(* for the test it's the parameter ``expiringTime`` *)
	expiring	:TIME;
END_VAR
VAR
	(* just the expectation if the assertion to test must be wrong or true *)
	assertionIsWrong		:BOOL;
	(* contains the format string for the test message *)
	message					:Tc2_System.T_MaxString;
	(* TwinCAT printf with the test message *)
	messageStringBuilder	:Tc2_Utilities.FB_FormatString;
	(* TIME value of ``expiringTime`` as string *)
	expiringTimeAsString	:STRING(22);
	(* TIME value of ``expectedValue`` as string *)
	timestampAsString		:STRING(22);
END_VAR
THIS^.assertorContainer.resetAssertor();

assertionIsWrong := (getTimePassed(startTime := valueToTest) > expiring);

message := SEL(
	assertionIsWrong,
	'timestamp is %s expiringTime is %s assertion must be TRUE', 
	'timestamp is %s expiringTime is %s assertion must be FALSE'
);
timestampAsString := TO_STRING(valueToTest);
expiringTimeAsString := TO_STRING(expiring);

messageStringBuilder(
	sFormat := message,
	arg1 := THIS^.AnyToArg(timestampAsString),
	arg2 := THIS^.AnyToArg(expiringTimeAsString)
);

THIS^.assertorContainer.assertor.assert.times.simple.timeHasNotExpired(
	timestamp		:= valueToTest,
	expiringTime	:= expiring,
	message			:= ''
);

THIS^.AssertEquals_BOOL(
	Expected 	:= assertionIsWrong,
	Actual 		:= THIS^.assertorContainer.wasAssertionWrong,
	Message 	:= messageStringBuilder.sOut
);
END_METHOD

(*

short summary
==================
This test method tests ``assert.times.simple.valueIsEqualTo``
method of CNM_AssertionInterfaces library, 
it provides the possibility to handover test data via parameter 


.. <legal notes>

legal notes
=================
| SPDX-FileCopyrightText: © 2022 ekvip automation GmbH <info@ekvip.de>
| SPDX-License-Identifier: Apache-2.0
| For details check: Apache-2.0_

.. _Apache-2.0: https://www.apache.org/licenses/LICENSE-2.0

.. </legal notes>

parameters
==========

*)

METHOD testValueIsEqualTo 
VAR_INPUT
	(* for the test it's the parameter ``currentValue`` *)
	valueToTest	:TIME;
	(* for the test it's the parameter ``expectedValue`` *)
	expected	:TIME;
END_VAR
VAR
	(* just the expectation if the assertion to test must be worng or true *)
	assertionIsWrong		:BOOL;
	(* contains the format string for the test message *)
	message					:Tc2_System.T_MaxString;
	(* TwinCAT printf with the test message *)
	messageStringBuilder	:Tc2_Utilities.FB_FormatString;
	(* TIME value of ``currentValue`` as string *)
	currentValueAsString	:STRING(22);
	(* TIME value of ``expectedValue`` as string *)
	expectedValueAsString	:STRING(22);
END_VAR
THIS^.assertorContainer.resetAssertor();

assertionIsWrong := (valueToTest <> expected);

message := SEL(
	assertionIsWrong,
	'currentValue is %s expectedValue is %s assertion must be TRUE', 
	'currentValue is %s expectedValue is %s assertion must be FALSE'
);
currentValueAsString := TO_STRING(valueToTest);
expectedValueAsString := TO_STRING(expected);

messageStringBuilder(
	sFormat := message,
	arg1 := THIS^.AnyToArg(currentValueAsString),
	arg2 := THIS^.AnyToArg(expectedValueAsString)
);

THIS^.assertorContainer.assertor.assert.times.simple.valueIsEqualTo(
	currentValue	:= valueToTest,
	expectedValue	:= expected,
	message			:= ''
);

THIS^.AssertEquals_BOOL(
	Expected 	:= assertionIsWrong,
	Actual 		:= THIS^.assertorContainer.wasAssertionWrong,
	Message 	:= messageStringBuilder.sOut
);
END_METHOD

(*

short summary
==================
This test method tests ``assert.times.simple.valueIsGreaterThan``
method of CNM_AssertionInterfaces library, 
it provides the possibility to handover test data via parameter 


.. <legal notes>

legal notes
=================
| SPDX-FileCopyrightText: © 2022 ekvip automation GmbH <info@ekvip.de>
| SPDX-License-Identifier: Apache-2.0
| For details check: Apache-2.0_

.. _Apache-2.0: https://www.apache.org/licenses/LICENSE-2.0

.. </legal notes>

parameters
==========

*)

METHOD testValueIsGreaterThan 
VAR_INPUT
	(* for the test it's the parameter ``currentValue`` *)
	valueToTest	:TIME;
	(* for the test it's the parameter ``lessValue`` *)
	lessValue	:TIME;
END_VAR
VAR
	(* just the expectation if the assertion to test must be worng or true *)
	assertionIsWrong		:BOOL;
	(* contains the format string for the test message *)
	message					:Tc2_System.T_MaxString;
	(* TwinCAT printf with the test message *)
	messageStringBuilder	:Tc2_Utilities.FB_FormatString;
	(* TIME value of ``currentValue`` as string *)
	currentValueAsString	:STRING(22);
	(* TIME value of ``lessValue`` as string *)
	lessValueAsString		:STRING(22);
END_VAR
THIS^.assertorContainer.resetAssertor();

assertionIsWrong := (valueToTest <= lessValue);

message := SEL(
	assertionIsWrong,
	'currentValue is %s lessValue is %s assertion must be TRUE', 
	'currentValue is %s lessValue is %s assertion must be FALSE'
);
currentValueAsString := TO_STRING(valueToTest);
lessValueAsString := TO_STRING(lessValue);

messageStringBuilder(
	sFormat := message,
	arg1 := THIS^.AnyToArg(currentValueAsString),
	arg2 := THIS^.AnyToArg(lessValueAsString)
);

THIS^.assertorContainer.assertor.assert.times.simple.valueIsGreaterThan(
	currentValue	:= valueToTest,
	lessValue		:= lessValue,
	message			:= ''
);

THIS^.AssertEquals_BOOL(
	Expected 	:= assertionIsWrong,
	Actual 		:= THIS^.assertorContainer.wasAssertionWrong,
	Message 	:= messageStringBuilder.sOut
);
END_METHOD

(*

short summary
==================
This test method tests ``assert.times.simple.valueIsInRangeOf``
method of CNM_AssertionInterfaces library, 
it provides the possibility to handover test data via parameter 


.. <legal notes>

legal notes
=================
| SPDX-FileCopyrightText: © 2022 ekvip automation GmbH <info@ekvip.de>
| SPDX-License-Identifier: Apache-2.0
| For details check: Apache-2.0_

.. _Apache-2.0: https://www.apache.org/licenses/LICENSE-2.0

.. </legal notes>

parameters
==========

*)

METHOD testValueIsInRangeOf 
VAR_INPUT
	(* for the test it's the parameter ``lowerLimit`` *)
	lowerLimit	:TIME;
	(* for the test it's the parameter ``currentValue`` *)
	valueToTest	:TIME;
	(* for the test it's the parameter ``upperLimit`` *)
	upperLimit	:TIME;
END_VAR
VAR
	(* just the expectation if the assertion to test must be worng or true *)
	assertionIsWrong		:BOOL;
	(* contains the format string for the test message *)
	message					:Tc2_System.T_MaxString;
	(* TwinCAT printf with the test message *)
	messageStringBuilder	:Tc2_Utilities.FB_FormatString;
	(* TIME value of ``lowerLimit`` as string *)
	lowerLimitAsString		:STRING(22);
	(* TIME value of ``currentValue`` as string *)
	currentValueAsString	:STRING(22);
	(* TIME value of ``upperLimit`` as string *)
	upperLimitAsString		:STRING(22);

END_VAR
THIS^.assertorContainer.resetAssertor();

assertionIsWrong := ((
		valueToTest < lowerLimit
	) OR (
		valueToTest > upperLimit
	)
);

message := SEL(
	assertionIsWrong,
	'lowerLimit is %s currentValue is %s upperLimit is %s assertion must be TRUE', 
	'lowerLimit is %s currentValue is %s upperLimit is %s assertion must be FALSE'
);
lowerLimitAsString		:= TO_STRING(lowerLimit);
currentValueAsString	:= TO_STRING(valueToTest);
upperLimitAsString		:= TO_STRING(upperLimit);

messageStringBuilder(
	sFormat := message,
	arg1 := THIS^.AnyToArg(lowerLimitAsString),
	arg2 := THIS^.AnyToArg(currentValueAsString),
	arg3 := THIS^.AnyToArg(upperLimitAsString)
);

THIS^.assertorContainer.assertor.assert.times.simple.valueIsInRangeOf(
	lowerLimit		:= lowerLimit,
	currentValue	:= valueToTest,
	upperLimit		:= upperLimit,
	message			:= ''
);

THIS^.AssertEquals_BOOL(
	Expected 	:= assertionIsWrong,
	Actual 		:= THIS^.assertorContainer.wasAssertionWrong,
	Message 	:= messageStringBuilder.sOut
);
END_METHOD

(*

short summary
==================
This test method tests ``assert.times.simple.valueIsLessThan``
method of CNM_AssertionInterfaces library, 
it provides the possibility to handover test data via parameter 


.. <legal notes>

legal notes
=================
| SPDX-FileCopyrightText: © 2022 ekvip automation GmbH <info@ekvip.de>
| SPDX-License-Identifier: Apache-2.0
| For details check: Apache-2.0_

.. _Apache-2.0: https://www.apache.org/licenses/LICENSE-2.0

.. </legal notes>

parameters
==========

*)

METHOD testValueIsLessThan 
VAR_INPUT
	(* for the test it's the parameter ``currentValue`` *)
	valueToTest		:TIME;
	(* for the test it's the parameter ``greaterValue`` *)
	greaterValue	:TIME;
END_VAR
VAR
	(* just the expectation if the assertion to test must be worng or true *)
	assertionIsWrong		:BOOL;
	(* contains the format string for the test message *)
	message					:Tc2_System.T_MaxString;
	(* TwinCAT printf with the test message *)
	messageStringBuilder	:Tc2_Utilities.FB_FormatString;
	(* TIME value of ``currentValue`` as string *)
	currentValueAsString	:STRING(22);
	(* TIME value of ``greaterValue`` as string *)
	greaterValueAsString	:STRING(22);
END_VAR
THIS^.assertorContainer.resetAssertor();

assertionIsWrong := (valueToTest >= greaterValue);

message := SEL(
	assertionIsWrong,
	'currentValue is %s greaterValue is %s assertion must be TRUE', 
	'currentValue is %s greaterValue is %s assertion must be FALSE'
);
currentValueAsString := TO_STRING(valueToTest);
greaterValueAsString := TO_STRING(greaterValue);

messageStringBuilder(
	sFormat := message,
	arg1 := THIS^.AnyToArg(currentValueAsString),
	arg2 := THIS^.AnyToArg(greaterValueAsString)
);

THIS^.assertorContainer.assertor.assert.times.simple.valueIsLessThan(
	currentValue	:= valueToTest,
	greaterValue	:= greaterValue,
	message			:= ''
);

THIS^.AssertEquals_BOOL(
	Expected 	:= assertionIsWrong,
	Actual 		:= THIS^.assertorContainer.wasAssertionWrong,
	Message 	:= messageStringBuilder.sOut
);
END_METHOD

(*

short summary
==================
This test method tests ``assert.times.simple.valueIsMax``
method of CNM_AssertionInterfaces library, 
it provides the possibility to handover test data via parameter 


.. <legal notes>

legal notes
=================
| SPDX-FileCopyrightText: © 2022 ekvip automation GmbH <info@ekvip.de>
| SPDX-License-Identifier: Apache-2.0
| For details check: Apache-2.0_

.. _Apache-2.0: https://www.apache.org/licenses/LICENSE-2.0

.. </legal notes>

parameters
==========

*)

METHOD testValueIsMax 
VAR_INPUT
	(* for the test it's the parameter ``currentValue`` *)
	valueToTest		:TIME;
	(* for the test it's the parameter ``greaterValue`` *)
	maximumValue	:TIME;
END_VAR
VAR
	(* just the expectation if the assertion to test must be worng or true *)
	assertionIsWrong		:BOOL;
	(* contains the format string for the test message *)
	message					:Tc2_System.T_MaxString;
	(* TwinCAT printf with the test message *)
	messageStringBuilder	:Tc2_Utilities.FB_FormatString;
	(* TIME value of ``currentValue`` as string *)
	currentValueAsString	:STRING(22);
	(* TIME value of ``maximumValue`` as string *)
	maximumValueAsString	:STRING(22);
END_VAR
THIS^.assertorContainer.resetAssertor();

assertionIsWrong := (valueToTest > maximumValue);

message := SEL(
	assertionIsWrong,
	'currentValue is %s maximumValue is %s assertion must be TRUE', 
	'currentValue is %s maximumValue is %s assertion must be FALSE'
);
currentValueAsString := TO_STRING(valueToTest);
maximumValueAsString := TO_STRING(maximumValue);

messageStringBuilder(
	sFormat := message,
	arg1 := THIS^.AnyToArg(currentValueAsString),
	arg2 := THIS^.AnyToArg(maximumValueAsString)
);

THIS^.assertorContainer.assertor.assert.times.simple.valueIsMax(
	currentValue	:= valueToTest,
	maximumValue	:= maximumValue,
	message			:= ''
);

THIS^.AssertEquals_BOOL(
	Expected 	:= assertionIsWrong,
	Actual 		:= THIS^.assertorContainer.wasAssertionWrong,
	Message 	:= messageStringBuilder.sOut
);
END_METHOD

(*

short summary
==================
This test method tests ``assert.times.simple.valueIsMin``
method of CNM_AssertionInterfaces library, 
it provides the possibility to handover test data via parameter 


.. <legal notes>

legal notes
=================
| SPDX-FileCopyrightText: © 2022 ekvip automation GmbH <info@ekvip.de>
| SPDX-License-Identifier: Apache-2.0
| For details check: Apache-2.0_

.. _Apache-2.0: https://www.apache.org/licenses/LICENSE-2.0

.. </legal notes>

parameters
==========

*)

METHOD testValueIsMin 
VAR_INPUT
	(* for the test it's the parameter ``currentValue`` *)
	valueToTest		:TIME;
	(* for the test it's the parameter ``greaterValue`` *)
	minimumValue	:TIME;
END_VAR
VAR
	(* just the expectation if the assertion to test must be worng or true *)
	assertionIsWrong		:BOOL;
	(* contains the format string for the test message *)
	message					:Tc2_System.T_MaxString;
	(* TwinCAT printf with the test message *)
	messageStringBuilder	:Tc2_Utilities.FB_FormatString;
	(* TIME value of ``currentValue`` as string *)
	currentValueAsString	:STRING(22);
	(* TIME value of ``minimumValue`` as string *)
	minimumValueAsString	:STRING(22);
END_VAR
THIS^.assertorContainer.resetAssertor();

assertionIsWrong := (valueToTest < minimumValue);

message := SEL(
	assertionIsWrong,
	'currentValue is %s minimumValue is %s assertion must be TRUE', 
	'currentValue is %s minimumValue is %s assertion must be FALSE'
);
currentValueAsString := TO_STRING(valueToTest);
minimumValueAsString := TO_STRING(minimumValue);

messageStringBuilder(
	sFormat := message,
	arg1 := THIS^.AnyToArg(currentValueAsString),
	arg2 := THIS^.AnyToArg(minimumValueAsString)
);

THIS^.assertorContainer.assertor.assert.times.simple.valueIsMin(
	currentValue	:= valueToTest,
	minimumValue	:= minimumValue,
	message			:= ''
);

THIS^.AssertEquals_BOOL(
	Expected 	:= assertionIsWrong,
	Actual 		:= THIS^.assertorContainer.wasAssertionWrong,
	Message 	:= messageStringBuilder.sOut
);
END_METHOD

(*

short summary
==================
This test method tests ``assert.times.simple.valueIsNotEqualTo``
method of CNM_AssertionInterfaces library, 
it provides the possibility to handover test data via parameter 


.. <legal notes>

legal notes
=================
| SPDX-FileCopyrightText: © 2022 ekvip automation GmbH <info@ekvip.de>
| SPDX-License-Identifier: Apache-2.0
| For details check: Apache-2.0_

.. _Apache-2.0: https://www.apache.org/licenses/LICENSE-2.0

.. </legal notes>

parameters
==========

*)

METHOD testValueIsNotEqualTo 
VAR_INPUT
	(* for the test it's the parameter ``currentValue`` *)
	valueToTest		:TIME;
	(* for the test it's the parameter ``unexpectedValue`` *)
	unexpectedValue	:TIME;
END_VAR
VAR
	(* just the expectation if the assertion to test must be worng or true *)
	assertionIsWrong		:BOOL;
	(* contains the format string for the test message *)
	message					:Tc2_System.T_MaxString;
	(* TwinCAT printf with the test message *)
	messageStringBuilder	:Tc2_Utilities.FB_FormatString;
	(* TIME value of ``currentValue`` as string *)
	currentValueAsString	:STRING(22);
	(* TIME value of ``unexpectedValue`` as string *)
	unexpectedValueAsString	:STRING(22);
END_VAR
THIS^.assertorContainer.resetAssertor();

assertionIsWrong := (valueToTest = unexpectedValue);

message := SEL(
	assertionIsWrong,
	'currentValue is %s expectedValue is %s assertion must be TRUE', 
	'currentValue is %s expectedValue is %s assertion must be FALSE'
);
currentValueAsString := TO_STRING(valueToTest);
unexpectedValueAsString := TO_STRING(unexpectedValue);

messageStringBuilder(
	sFormat := message,
	arg1 := THIS^.AnyToArg(currentValueAsString),
	arg2 := THIS^.AnyToArg(unexpectedValueAsString)
);

THIS^.assertorContainer.assertor.assert.times.simple.valueIsNotEqualTo(
	currentValue	:= valueToTest,
	unexpectedValue	:= unexpectedValue,
	message			:= ''
);

THIS^.AssertEquals_BOOL(
	Expected 	:= assertionIsWrong,
	Actual 		:= THIS^.assertorContainer.wasAssertionWrong,
	Message 	:= messageStringBuilder.sOut
);
END_METHOD

END_FUNCTION_BLOCK

// ---- AssertionTester/classes/AssertionTester.TcPOU
(*

short summary
=============

.. <legal notes>

legal notes
=================
| SPDX-FileCopyrightText: © 2023 ekvip automation GmbH <info@ekvip.de>
| SPDX-License-Identifier: Apache-2.0
| For details check: Apache-2.0_

.. _Apache-2.0: https://www.apache.org/licenses/LICENSE-2.0

.. </legal notes>

methods and properties
======================

*)


FUNCTION_BLOCK AssertionTester EXTENDS CNM_AbstractObject.Object IMPLEMENTS IAttachAssertorContainer
VAR	
	pointerTests 			:PointerAssertionsTests(classToBeTested := 0);
	uxintAssertions			:UxintAssertionTests(classToBeTested := 0);
	usintAssertions			:UsintAssertionTests(classToBeTested := 0);
	uintAssertions			:UintAssertionTests(classToBeTested := 0);
	udintAssertions			:UdintAssertionTests(classToBeTested := 0);
	ulintAssertions			:UlintAssertionTests(classToBeTested := 0);	
	xintAssertions			:XintAssertionTests(classToBeTested := 0);
	sintAssertions			:SintAssertionTests(classToBeTested := 0);
	intAssertions			:IntAssertionTests(classToBeTested := 0);
	dintAssertions			:DintAssertionTests(classToBeTested := 0);
	lintAssertions			:LintAssertionTests(classToBeTested := 0);
	lrealAssertions		 	:LRealAssertionTests(classToBeTested := 0);
	realAssertions			:RealAssertionTests(classToBeTested := 0);
	bitNumberAssertiosByte	:ByteAssertionTests(classToBeTested := 0);
	bitNumberAssertionsWord :WordAssertionTests(classToBeTested := 0);
	bitNumberAssertionDword	:DWordAssertionTests(classToBeTested := 0);
	bitNumberAssertionLWord :LWordAssertionTests(classToBeTested := 0);
	bitNumberAssertionXWord :XWordAssertionTests(classToBeTested := 0);
	binaryTests				:BinaryAssertionsTests(classToBeTested := 0);
	dateAndTimeAssertions 	:DTAssertionTests(classToBeTested := 0);
	ldateAndTimeAssertions 	:LDTAssertionTests(classToBeTested := 0);
	timeTests				:TimeAssertionsTests(classToBeTested := 0);
	ltimeTests				:LTimeAssertionsTests(classToBeTested := 0);
	windows125xStringTests	:Windows125xStringAssertionTests(classToBeTested := 0);
	unicodeUtf8StringTests	:UnicodeUtf8StringAssertionTests(classToBeTested := 0);
	unicodeUtf16StringTests	:UnicodeUtf16StringAssertionTests(classToBeTested := 0);
	objectTests				:ObjectAssertionsTests(classToBeTested := 0);
	dateAssertions			:DateAssertionTests(classToBeTested := 0);
	ldateAssertions			:LDateAssertionTests(classToBeTested := 0);
	timeOfDayAssertions 	:TODAssertionTests(classToBeTested := 0);
	ltimeOfDayAssertions 	:LTODAssertionTests(classToBeTested := 0);
END_VAR

(*

short summary
=============

.. <legal notes>

legal notes
=================
| SPDX-FileCopyrightText: © 2023 ekvip automation GmbH <info@ekvip.de>
| SPDX-License-Identifier: Apache-2.0
| For details check: Apache-2.0_

.. _Apache-2.0: https://www.apache.org/licenses/LICENSE-2.0

.. </legal notes>

*)

PROPERTY attachAssertorContainer : IAssertorContainer
SET

THIS^.timeTests.attachAssertorContainer					:= attachAssertorContainer;
THIS^.ltimeTests.attachAssertorContainer				:= attachAssertorContainer;
THIS^.windows125xStringTests.attachAssertorContainer	:= attachAssertorContainer;
THIS^.unicodeUtf8StringTests.attachAssertorContainer	:= attachAssertorContainer;
THIS^.unicodeUtf16StringTests.attachAssertorContainer	:= attachAssertorContainer;
THIS^.objectTests.attachAssertorContainer 				:= attachAssertorContainer;
THIS^.pointerTests.attachAssertorContainer 				:= attachAssertorContainer;
THIS^.binaryTests.attachAssertorContainer 				:= attachAssertorContainer;
THIS^.lrealAssertions.attachAssertorContainer 			:= attachAssertorContainer;
THIS^.realAssertions.attachAssertorContainer 			:= attachAssertorContainer;
THIS^.dateAssertions.attachAssertorContainer 			:= attachAssertorContainer;
THIS^.ldateAssertions.attachAssertorContainer 			:= attachAssertorContainer;
THIS^.dateAndTimeAssertions.attachAssertorContainer		:= attachAssertorContainer;
THIS^.ldateAndTimeAssertions.attachAssertorContainer	:= attachAssertorContainer;
THIS^.timeOfDayAssertions.attachAssertorContainer		:= attachAssertorContainer;
THIS^.ltimeOfDayAssertions.attachAssertorContainer		:= attachAssertorContainer;
THIS^.usintAssertions.attachAssertorContainer			:= attachAssertorContainer;
THIS^.uintAssertions.attachAssertorContainer			:= attachAssertorContainer;
THIS^.udintAssertions.attachAssertorContainer			:= attachAssertorContainer;
THIS^.ulintAssertions.attachAssertorContainer			:= attachAssertorContainer;
THIS^.uxintAssertions.attachAssertorContainer			:= attachAssertorContainer;
THIS^.sintAssertions.attachAssertorContainer			:= attachAssertorContainer;
THIS^.intAssertions.attachAssertorContainer				:= attachAssertorContainer;
THIS^.dintAssertions.attachAssertorContainer			:= attachAssertorContainer;
THIS^.lintAssertions.attachAssertorContainer			:= attachAssertorContainer;
THIS^.xintAssertions.attachAssertorContainer			:= attachAssertorContainer;
THIS^.bitNumberAssertiosByte.attachAssertorContainer	:= attachAssertorContainer;
THIS^.bitNumberAssertionsWord.attachAssertorContainer	:= attachAssertorContainer;
THIS^.bitNumberAssertionDword.attachAssertorContainer	:= attachAssertorContainer;
THIS^.bitNumberAssertionLWord.attachAssertorContainer	:= attachAssertorContainer;
THIS^.bitNumberAssertionXWord.attachAssertorContainer	:= attachAssertorContainer;
END_SET
END_PROPERTY

(*

short summary
=============

.. <legal notes>

legal notes
=================
| SPDX-FileCopyrightText: © 2023 ekvip automation GmbH <info@ekvip.de>
| SPDX-License-Identifier: Apache-2.0
| For details check: Apache-2.0_

.. _Apache-2.0: https://www.apache.org/licenses/LICENSE-2.0

.. </legal notes>

*)

PROPERTY className :CNM_AbstractObject.ClassName
GET
(*

short summary
=============

.. <legal notes>

legal notes
=================
| SPDX-FileCopyrightText: © 2023 ekvip automation GmbH <info@ekvip.de>
| SPDX-License-Identifier: Apache-2.0
| For details check: Apache-2.0_

.. _Apache-2.0: https://www.apache.org/licenses/LICENSE-2.0

.. </legal notes>

*)

VAR
END_VAR
className := 'AssertionTester';
END_GET
END_PROPERTY

(*

short summary
=================
The constructor ``FB_init`` is needed to create an unique hash code.
The hash code is a pseudo random number create with a xorshift_ algorithm.
It can be overwritten on derivations, because it will be called implicit, ``SUPER^.FB_init()`` is not required.
For more information check: `Behavoir with derived function blocks`_

.. _Behavoir with derived function blocks: https://infosys.beckhoff.com/content/1033/tc3_plc_intro/5482088715.html?id=6983869892358031022
.. _xorshift: https://en.wikipedia.org/wiki/Xorshift

.. <legal notes>

legal notes
=================
| SPDX-FileCopyrightText: © 2022 ekvip automation GmbH <info@ekvip.de>
| SPDX-License-Identifier: Apache-2.0
| For details check: Apache-2.0_

.. _Apache-2.0: https://www.apache.org/licenses/LICENSE-2.0

.. </legal notes>

parameters
=================

*)

METHOD FB_init :BOOL
VAR_INPUT
	(* if TRUE, the retain variables are initialized (warm start / cold start)*)
	bInitRetains	:BOOL;
	(* if TRUE, the instance afterwards gets moved into the copy code (online change) *)
	bInCopyCode		:BOOL;
	(* assertor class to test *)
	classToBeTested :IAssertorContainer;
END_VAR
VAR
	{attribute 'hide'}
	newHashstate3		:CNM_AbstractObject.Hashcode;
END_VAR
VAR CONSTANT
	{attribute 'hide'}
	NUMBER_OF_LEFT_SHIFTS		:UINT	:= 17;
	{attribute 'hide'}
	NUMBER_OF_LEFT_ROTATIONS	:UINT   := 45;
END_VAR
THIS^.attachAssertorContainer := classToBeTested;
END_METHOD

END_FUNCTION_BLOCK

// ---- Project Information/F_GetCompany.TcPOU
// This function has been automatically generated from the project information.
{attribute 'signature_flag' := '1073741824'}
{attribute 'TcGenerated'}
{attribute 'no-analysis'}
FUNCTION F_GetCompany : WSTRING
VAR_INPUT
	
END_VAR

F_GetCompany := "ekvip automation GmbH";

END_FUNCTION

// ---- Project Information/F_GetTitle.TcPOU
// This function has been automatically generated from the project information.
{attribute 'signature_flag' := '1073741824'}
{attribute 'TcGenerated'}
{attribute 'no-analysis'}
FUNCTION F_GetTitle : WSTRING
VAR_INPUT
	
END_VAR

F_GetTitle := "CNM_AssertionInterfaceTests";

END_FUNCTION

// ---- Project Information/F_GetVersion.TcPOU
// This function has been automatically generated from the project information.
{attribute 'signature_flag' := '1073741824'}
{attribute 'TcGenerated'}
{attribute 'no-analysis'}
FUNCTION F_GetVersion : ST_LibVersion
VAR_INPUT
	
END_VAR

F_GetVersion.iMajor := 1;
F_GetVersion.iMinor := 2;
F_GetVersion.iBuild := 0;
F_GetVersion.iRevision := 6;
F_GetVersion.sVersion := '1.2.0.6';
F_GetVersion.nFlags := 0;

END_FUNCTION

// ---- AssertionTester/AssertionTests/BitNumberAssertions/classes/XWordAssertionTests.TcPOU
(*

x summary
==================
This class tests all methods of __XWORD assertions
with various combinations of inputs and checks expected 
outputs are satisfied or not

.. <legal notes>

legal notes
=================
| SPDX-FileCopyrightText: © 2022 ekvip automation GmbH <info@ekvip.de>
| SPDX-License-Identifier: Apache-2.0
| For details check: Apache-2.0_

.. _Apache-2.0: https://www.apache.org/licenses/LICENSE-2.0

.. </legal notes>

methods and properties
======================

*)

FUNCTION_BLOCK XWordAssertionTests EXTENDS AbstractAssertorTest
VAR_INPUT
END_VAR
VAR CONSTANT
	(* number of the lsb *)
	FIRST_BIT				:USINT := 0;
	(* number of the msb *)
	LAST_BIT				:USINT := ((SIZEOF(__XWORD)*8)-1);
	(* just the value zero *)
	ZERO					:__XINT := 0;
	(* no single bit is set, it's just the value zero *)
	NO_BIT_SET				:__XWORD := 0;
	(* just the lsb is set, it's just the value one *)
	LSB_ONLY				:__XWORD := 1;
	(* all bits are set *)
	ALL_BITS_SET			:__XWORD := (NOT NO_BIT_SET);
	(* the msb is set only *)
	MSB_ONLY				:__XWORD := ROR(LSB_ONLY,1);
	(* prefix to unify the test names *)
	TEST_NAME_PREFIX		:STRING := 'assert.bitNumber.x.';
	(* number how many times the product will be rotated right *)
	NUMBER_OF_RORS			:__UXINT := 1;
	(* multiplicand for the ``multiplier`` *)
	MULTIPLICAND			:__UXINT := 16#1111_1111;
	(* first of all multipliers the test iterates *)
	FIRST_MULTIPLIER		:__UXINT := 0;
	(* first of all multipliers the test iterates *)
	LAST_MULTIPLIER			:__UXINT := 15;
	(* constant for the modulo operator to check if valueToTest is even (lsb is unset) or odd (lsb is set) *)
	DEVISOR_FOR_EVEN_ODD	:__UXINT := 2;
END_VAR

THIS^.runAndMaskIsEqualToTests();
THIS^.runAndMaskIsNotEqualToTests();
THIS^.runBitXIsEqualToTests();
THIS^.runBitXIsNotEqualToTests();
THIS^.runBitXIsSetTests();
THIS^.runBitXIsUnsetTests();
THIS^.runLsbIsEqualToTests();
THIS^.runLsbIsNotEqualToTests();
THIS^.runLsbIsSetTests();
THIS^.runLsbIsUnsetTests();
THIS^.runMsbIsEqualToTests();
THIS^.runMsbIsNotEqualToTests();
THIS^.runMsbIsSetTests();
THIS^.runMsbIsUnsetTests();
THIS^.runOrMaskIsEqualToTests();
THIS^.runOrMaskIsNotEqualToTests();
THIS^.runValueIsMaxTests();
THIS^.runValueIsMinTests();
THIS^.runValueIsEqualToTests();
THIS^.runValueIsGreaterTests();
THIS^.runValueIsLessThanTests();
THIS^.runValueIsInRangeOfTests();
THIS^.runValueIsNotEqualToTests();
THIS^.runXorMaskIsEqualToTests();
THIS^.runXorMaskIsNotEqualToTests();

(*

x summary
==================
This test method is a helper function to create a unified test name

.. <legal notes>

legal notes
=================
| SPDX-FileCopyrightText: © 2022 ekvip automation GmbH <info@ekvip.de>
| SPDX-License-Identifier: Apache-2.0
| For details check: Apache-2.0_

.. _Apache-2.0: https://www.apache.org/licenses/LICENSE-2.0

.. </legal notes>

parameters
==========

*)

METHOD PROTECTED getTestNameFor :Tc2_System.T_MaxString
VAR_INPUT
	(* name of the method to test, to create a unified test name *)
	nameOfMethodToTest	:Tc2_System.T_MaxString;
END_VAR
getTestNameFor := Tc2_Standard.CONCAT(THIS^.TEST_NAME_PREFIX, nameOfMethodToTest);
END_METHOD

(*

x summary
==================
This test method tests ``assert.bitNumber.x.andMaskIsEqualTo``
method of CNM_AssertionInterfaces library with various inputs

.. <legal notes>

legal notes
=================
| SPDX-FileCopyrightText: © 2022 ekvip automation GmbH <info@ekvip.de>
| SPDX-License-Identifier: Apache-2.0
| For details check: Apache-2.0_

.. _Apache-2.0: https://www.apache.org/licenses/LICENSE-2.0

.. </legal notes>

*)

METHOD runAndMaskIsEqualToTests
VAR
	(* shift to iterate through the bit numbers *)
	shift				:__UXINT;
	(* mask with the bit iteration *)
	mask				:__XWORD;
END_VAR
RETURN (NOT TcUnit.TEST_ORDERED(THIS^.getTestNameFor('AndMaskIsEqualTo')));

FOR shift:= THIS^.FIRST_BIT TO THIS^.LAST_BIT DO
	mask := SHL(THIS^.LSB_ONLY, shift);
	THIS^.testAndMaskIsEqualTo(
		valueToTest := THIS^.ALL_BITS_SET,
		mask  := mask,
		expected := mask
	);
	THIS^.testAndMaskIsEqualTo(
		valueToTest := THIS^.ALL_BITS_SET,
		mask  := mask,
		expected := (NOT mask)
	);
	THIS^.testAndMaskIsEqualTo(
		valueToTest := mask,
		mask  := (NOT mask),
		expected := THIS^.NO_BIT_SET
	);
	THIS^.testAndMaskIsEqualTo(
		valueToTest := mask,
		mask  := (NOT mask),
		expected := (NOT mask)
	);	
	THIS^.testAndMaskIsEqualTo(
		valueToTest := mask,
		mask  := mask,
		expected := mask
	);	
END_FOR

THIS^.testAndMaskIsEqualTo(
	valueToTest := THIS^.NO_BIT_SET,
	mask  := THIS^.NO_BIT_SET,
	expected := THIS^.NO_BIT_SET
);
THIS^.testAndMaskIsEqualTo(
	valueToTest := THIS^.NO_BIT_SET,
	mask  := THIS^.NO_BIT_SET,
	expected := THIS^.LSB_ONLY
);

THIS^.testAndMaskIsEqualTo(
	valueToTest := THIS^.ALL_BITS_SET,
	mask  := THIS^.ALL_BITS_SET,
	expected := THIS^.ALL_BITS_SET
);
THIS^.testAndMaskIsEqualTo(
	valueToTest := THIS^.ALL_BITS_SET,
	mask  := THIS^.ALL_BITS_SET,
	expected := THIS^.NO_BIT_SET
);

TcUnit.TEST_FINISHED();
END_METHOD

(*

x summary
==================
This test method tests ``assert.bitNumber.x.andMaskIsNotEqualTo``
method of CNM_AssertionInterfaces library with various inputs

.. <legal notes>

legal notes
=================
| SPDX-FileCopyrightText: © 2022 ekvip automation GmbH <info@ekvip.de>
| SPDX-License-Identifier: Apache-2.0
| For details check: Apache-2.0_

.. _Apache-2.0: https://www.apache.org/licenses/LICENSE-2.0

.. </legal notes>

*)

METHOD runAndMaskIsNotEqualToTests
VAR
	(* shift to iterate through the bit numbers *)
	shift	:__UXINT;
	(* mask with the bit iteration *)
	mask	:__XWORD;
END_VAR
RETURN (NOT TcUnit.TEST_ORDERED(THIS^.getTestNameFor('AndMaskIsNotEqualTo')));

FOR shift:= THIS^.FIRST_BIT TO THIS^.LAST_BIT DO
	mask := SHL(THIS^.LSB_ONLY, shift);
	THIS^.testAndMaskIsNotEqualTo(
		valueToTest := THIS^.ALL_BITS_SET,
		mask  := mask,
		unexpected := (NOT mask)
	);
	THIS^.testAndMaskIsNotEqualTo(
		valueToTest := THIS^.ALL_BITS_SET,
		mask  := mask,
		unexpected := mask
	);
	THIS^.testAndMaskIsNotEqualTo(
		valueToTest := mask,
		mask  := (NOT mask),
		unexpected := (NOT mask)
	);	
	THIS^.testAndMaskIsNotEqualTo(
		valueToTest := mask,
		mask  := (NOT mask),
		unexpected := THIS^.NO_BIT_SET
	);
	THIS^.testAndMaskIsNotEqualTo(
		valueToTest := mask,
		mask  := mask,
		unexpected := mask
	);	
END_FOR

THIS^.testAndMaskIsNotEqualTo(
	valueToTest := THIS^.NO_BIT_SET,
	mask  := THIS^.NO_BIT_SET,
	unexpected := THIS^.LSB_ONLY
);
THIS^.testAndMaskIsNotEqualTo(
	valueToTest := THIS^.NO_BIT_SET,
	mask  := THIS^.NO_BIT_SET,
	unexpected := THIS^.NO_BIT_SET
);

THIS^.testAndMaskIsNotEqualTo(
	valueToTest := THIS^.ALL_BITS_SET,
	mask  := THIS^.ALL_BITS_SET,
	unexpected := THIS^.NO_BIT_SET
);
THIS^.testAndMaskIsNotEqualTo(
	valueToTest := THIS^.ALL_BITS_SET,
	mask  := THIS^.ALL_BITS_SET,
	unexpected := THIS^.ALL_BITS_SET
);

TcUnit.TEST_FINISHED();
END_METHOD

(*

x summary
==================
This test method tests ``assert.bitNumber.x.bitXIsEqualTo``
method of CNM_AssertionInterfaces library with various inputs

.. <legal notes>

legal notes
=================
| SPDX-FileCopyrightText: © 2022 ekvip automation GmbH <info@ekvip.de>
| SPDX-License-Identifier: Apache-2.0
| For details check: Apache-2.0_

.. _Apache-2.0: https://www.apache.org/licenses/LICENSE-2.0

.. </legal notes>

*)

METHOD runBitXIsEqualToTests
VAR
	(* this is the number of the bit to test *)
	bitNumberToTest	:CNM_AssertionInterfaces.BitNumberXWord;
	(* it's just part of the test data *)
	valueToTest		:__XWORD;
END_VAR
RETURN (NOT TcUnit.TEST_ORDERED(THIS^.getTestNameFor('bitXIsEqualTo')));

FOR bitNumberToTest := THIS^.FIRST_BIT TO THIS^.LAST_BIT DO

	valueToTest := SHL(THIS^.LSB_ONLY,bitNumberToTest);
	THIS^.testBitXIsEqualTo(
		valueToTest			:=valueToTest,
		bitNumberToCheck	:=bitNumberToTest,
		bitIsSet			:=TRUE
	);
	THIS^.testBitXIsEqualTo(
		valueToTest			:=valueToTest,
		bitNumberToCheck	:=bitNumberToTest,
		bitIsSet			:=FALSE
	);

	valueToTest := (NOT valueToTest);
	THIS^.testBitXIsEqualTo(
		valueToTest			:=valueToTest,
		bitNumberToCheck	:=bitNumberToTest,
		bitIsSet			:=FALSE
	);
	THIS^.testBitXIsEqualTo(
		valueToTest			:=valueToTest,
		bitNumberToCheck	:=bitNumberToTest,
		bitIsSet			:=TRUE
	);	
END_FOR

TcUnit.TEST_FINISHED();
END_METHOD

(*

x summary
==================
This test method tests ``assert.bitNumber.x.bitXIsNotEqualTo``
method of CNM_AssertionInterfaces library with various inputs

.. <legal notes>

legal notes
=================
| SPDX-FileCopyrightText: © 2022 ekvip automation GmbH <info@ekvip.de>
| SPDX-License-Identifier: Apache-2.0
| For details check: Apache-2.0_

.. _Apache-2.0: https://www.apache.org/licenses/LICENSE-2.0

.. </legal notes>

*)

METHOD runBitXIsNotEqualToTests
VAR
	(* this is the number of the bit to test *)
	bitNumberToTest	:CNM_AssertionInterfaces.BitNumberXWord;
	(* it's just part of the test data *)
	valueToTest		:__XWORD;
END_VAR
RETURN (NOT TcUnit.TEST_ORDERED(THIS^.getTestNameFor('bitXIsNotEqualTo')));

FOR bitNumberToTest := THIS^.FIRST_BIT TO THIS^.LAST_BIT DO
	valueToTest := SHL(THIS^.LSB_ONLY,bitNumberToTest);
	THIS^.testBitXIsNotEqualTo(
		valueToTest			:=valueToTest,
		bitNumberToCheck	:=bitNumberToTest,
		bitIsSet			:=TRUE
	);
	THIS^.testBitXIsNotEqualTo(
		valueToTest			:=valueToTest,
		bitNumberToCheck	:=bitNumberToTest,
		bitIsSet			:=FALSE
	);

	valueToTest := (NOT valueToTest);
	THIS^.testBitXIsNotEqualTo(
		valueToTest			:=valueToTest,
		bitNumberToCheck	:=bitNumberToTest,
		bitIsSet			:=TRUE
	);
	THIS^.testBitXIsNotEqualTo(
		valueToTest			:=valueToTest,
		bitNumberToCheck	:=bitNumberToTest,
		bitIsSet			:=FALSE
	);	
END_FOR

TcUnit.TEST_FINISHED();
END_METHOD

(*

x summary
==================
This test method tests ``assert.bitNumber.x.bitXIsSet`` 
of CNM_AssertionInterfaces library with various inputs

.. <legal notes>

legal notes
=================
| SPDX-FileCopyrightText: © 2022 ekvip automation GmbH <info@ekvip.de>
| SPDX-License-Identifier: Apache-2.0
| For details check: Apache-2.0_

.. _Apache-2.0: https://www.apache.org/licenses/LICENSE-2.0

.. </legal notes>

*)

METHOD runBitXIsSetTests
VAR
	(* this is the number of the bit to test *)
	bitNumberToTest	:CNM_AssertionInterfaces.BitNumberXWord;
	(* it's just part of the test data *)
	valueToTest		:__XWORD;
END_VAR
RETURN (NOT TcUnit.TEST_ORDERED(THIS^.getTestNameFor('bitXIsSet')));

FOR bitNumberToTest := THIS^.FIRST_BIT TO THIS^.LAST_BIT DO
	valueToTest := SHL(THIS^.LSB_ONLY,bitNumberToTest);
	THIS^.testBitXIsSet(
		valueToTest := valueToTest,
		bitNumberToCheck := bitNumberToTest
	);
	THIS^.testBitXIsSet(
		valueToTest := (NOT valueToTest),
		bitNumberToCheck := bitNumberToTest
	);
	THIS^.testBitXIsSet(
		valueToTest := THIS^.NO_BIT_SET,
		bitNumberToCheck := bitNumberToTest
	);
	THIS^.testBitXIsSet(
		valueToTest := THIS^.ALL_BITS_SET,
		bitNumberToCheck := bitNumberToTest
	);
END_FOR

TcUnit.TEST_FINISHED();
END_METHOD

(*

x summary
==================
This test method tests ``assert.bitNumber.x.bitXIsUnset``
of CNM_AssertionInterfaces library with various inputs

.. <legal notes>

legal notes
=================
| SPDX-FileCopyrightText: © 2022 ekvip automation GmbH <info@ekvip.de>
| SPDX-License-Identifier: Apache-2.0
| For details check: Apache-2.0_

.. _Apache-2.0: https://www.apache.org/licenses/LICENSE-2.0

.. </legal notes>

*)

METHOD runBitXIsUnsetTests
VAR
	(* this is the number of the bit to test *)
	bitNumberToTest	:CNM_AssertionInterfaces.BitNumberXWord;
	(* it's just part of the test data *)
	valueToTest		:__XWORD;
END_VAR
RETURN (NOT TcUnit.TEST_ORDERED(THIS^.getTestNameFor('bitXIsUnset')));

FOR bitNumberToTest := THIS^.FIRST_BIT TO THIS^.LAST_BIT DO
	valueToTest := SHL(THIS^.LSB_ONLY,bitNumberToTest);
	THIS^.testBitXIsUnset(
		valueToTest := valueToTest,
		bitNumberToCheck := bitNumberToTest
	);
	THIS^.testBitXIsUnset(
		valueToTest := (NOT valueToTest),
		bitNumberToCheck := bitNumberToTest
	);
	THIS^.testBitXIsUnset(
		valueToTest := THIS^.NO_BIT_SET,
		bitNumberToCheck := bitNumberToTest
	);
	THIS^.testBitXIsUnset(
		valueToTest :=THIS^.ALL_BITS_SET,
		bitNumberToCheck := bitNumberToTest
	);
END_FOR

TcUnit.TEST_FINISHED();
END_METHOD

(*

x summary
==================
This test method tests ``assert.bitNumber.x.lsbIsEqualTo``
method of CNM_AssertionInterfaces library with various inputs

.. <legal notes>

legal notes
=================
| SPDX-FileCopyrightText: © 2022 ekvip automation GmbH <info@ekvip.de>
| SPDX-License-Identifier: Apache-2.0
| For details check: Apache-2.0_

.. _Apache-2.0: https://www.apache.org/licenses/LICENSE-2.0

.. </legal notes>

*)

METHOD runLsbIsEqualToTests
VAR
	(* it's just part of the test data *)
	valueToTest	:__XWORD;
	(* multiplier to get various bit patterns *)
	multiplier	:__UXINT;
END_VAR
RETURN (NOT TcUnit.TEST_ORDERED(THIS^.getTestNameFor('lsbIsEqualTo')));

FOR multiplier := THIS^.FIRST_MULTIPLIER TO THIS^.LAST_MULTIPLIER DO
	valueToTest := (THIS^.MULTIPLICAND * multiplier);

	THIS^.testLsbIsEqualTo(
		valueToTest := valueToTest,
		expectedValue := TRUE
	);	
	THIS^.testLsbIsEqualTo(
		valueToTest := valueToTest,
		expectedValue := FALSE
	);

END_FOR

THIS^.testLsbIsEqualTo(
	valueToTest := THIS^.LSB_ONLY,
	expectedValue := TRUE
);	
THIS^.testLsbIsEqualTo(
	valueToTest := THIS^.LSB_ONLY,
	expectedValue := FALSE
);
THIS^.testLsbIsEqualTo(
	valueToTest := THIS^.MSB_ONLY,
	expectedValue := TRUE
);	
THIS^.testLsbIsEqualTo(
	valueToTest := THIS^.MSB_ONLY,
	expectedValue := FALSE
);

TcUnit.TEST_FINISHED();
END_METHOD

(*

x summary
==================
This test method tests ``assert.bitNumber.x.lsbIsNotEqualTo``
method of CNM_AssertionInterfaces library with various inputs

.. <legal notes>

legal notes
=================
| SPDX-FileCopyrightText: © 2022 ekvip automation GmbH <info@ekvip.de>
| SPDX-License-Identifier: Apache-2.0
| For details check: Apache-2.0_

.. _Apache-2.0: https://www.apache.org/licenses/LICENSE-2.0

.. </legal notes>

*)

METHOD runLsbIsNotEqualToTests
VAR
	(* it's just part of the test data *)
	valueToTest	:__XWORD;
	(* multiplier to get various bit patterns *)
	multiplier	:__UXINT;
END_VAR
RETURN (NOT TcUnit.TEST_ORDERED(THIS^.getTestNameFor('lsbIsNotEqualTo')));

FOR multiplier := THIS^.FIRST_MULTIPLIER TO THIS^.LAST_MULTIPLIER DO
	valueToTest := (THIS^.MULTIPLICAND * multiplier);

	THIS^.testLsbIsNotEqualTo(
		valueToTest := valueToTest,
		unexpectedValue := TRUE
	);	
	THIS^.testLsbIsNotEqualTo(
		valueToTest := valueToTest,
		unexpectedValue := FALSE
	);

END_FOR

THIS^.testLsbIsNotEqualTo(
	valueToTest := THIS^.LSB_ONLY,
	unexpectedValue := TRUE
);	
THIS^.testLsbIsNotEqualTo(
	valueToTest := THIS^.LSB_ONLY,
	unexpectedValue := FALSE
);
THIS^.testLsbIsNotEqualTo(
	valueToTest := THIS^.MSB_ONLY,
	unexpectedValue := TRUE
);	
THIS^.testLsbIsNotEqualTo(
	valueToTest := THIS^.MSB_ONLY,
	unexpectedValue := FALSE
);

TcUnit.TEST_FINISHED();
END_METHOD

(*

x summary
==================
This test method tests ``assert.bitNumber.x.lsbIsSet``
of CNM_AssertionInterfaces library with various inputs

.. <legal notes>

legal notes
=================
| SPDX-FileCopyrightText: © 2022 ekvip automation GmbH <info@ekvip.de>
| SPDX-License-Identifier: Apache-2.0
| For details check: Apache-2.0_

.. _Apache-2.0: https://www.apache.org/licenses/LICENSE-2.0

.. </legal notes>

*)

METHOD runLsbIsSetTests
VAR
	(* it's just part of the test data *)
	valueToTest	:__XWORD;
	(* multiplier to get various bit patterns *)
	multiplier	:__UXINT;
END_VAR
RETURN (NOT TcUnit.TEST_ORDERED(THIS^.getTestNameFor('lsbIsSet')));

FOR multiplier := THIS^.FIRST_MULTIPLIER TO THIS^.LAST_MULTIPLIER DO
	valueToTest := (THIS^.MULTIPLICAND * multiplier);
	THIS^.testLsbIsSet(
		valueToTest := valueToTest
	);
END_FOR

THIS^.testLsbIsSet(
	valueToTest := THIS^.MSB_ONLY
);	
THIS^.testLsbIsSet(
	valueToTest := THIS^.MSB_ONLY
);

TcUnit.TEST_FINISHED();
END_METHOD

(*

x summary
==================
This test method tests ``assert.bitNumber.x.lsbIsUnset``
of CNM_AssertionInterfaces library with various inputs

.. <legal notes>

legal notes
=================
| SPDX-FileCopyrightText: © 2022 ekvip automation GmbH <info@ekvip.de>
| SPDX-License-Identifier: Apache-2.0
| For details check: Apache-2.0_

.. _Apache-2.0: https://www.apache.org/licenses/LICENSE-2.0

.. </legal notes>

*)

METHOD runLsbIsUnsetTests
VAR
	(* it's just part of the test data *)
	valueToTest	:__XWORD;
	(* multiplier to get various bit patterns *)
	multiplier	:__UXINT;
END_VAR
RETURN (NOT TcUnit.TEST_ORDERED(THIS^.getTestNameFor('lsbIsUnset')));

FOR multiplier := THIS^.FIRST_MULTIPLIER TO THIS^.LAST_MULTIPLIER DO
	valueToTest := (THIS^.MULTIPLICAND * multiplier);
	THIS^.testLsbIsUnset(
		valueToTest := valueToTest
	);
END_FOR

THIS^.testLsbIsUnset(
	valueToTest := THIS^.LSB_ONLY
);	
THIS^.testLsbIsUnset(
	valueToTest := THIS^.MSB_ONLY
);

TcUnit.TEST_FINISHED();
END_METHOD

(*

x summary
==================
This test method tests ``assert.bitNumber.x.msbIsEqualTo``
method of CNM_AssertionInterfaces library with various inputs

.. <legal notes>

legal notes
=================
| SPDX-FileCopyrightText: © 2022 ekvip automation GmbH <info@ekvip.de>
| SPDX-License-Identifier: Apache-2.0
| For details check: Apache-2.0_

.. _Apache-2.0: https://www.apache.org/licenses/LICENSE-2.0

.. </legal notes>

*)

METHOD runMsbIsEqualToTests
VAR
	(* it's just part of the test data *)
	valueToTest	:__XWORD;
	(* multiplier to get various bit patterns *)
	multiplier	:__UXINT;
END_VAR
VAR CONSTANT
	(* number how many times the product will be rotated right *)
	NUMBER_OF_RORS :__UXINT := 1;
	(* multiplicand for the ``multiplier`` *)
	MULTIPLICAND :__UXINT := 17;
	(* first of all multipliers the test iterates *)
	FIRST_MULTIPLIER :__UXINT := 0;
	(* first of all multipliers the test iterates *)
	LAST_MULTIPLIER :__UXINT := 15;
END_VAR
RETURN (NOT TcUnit.TEST_ORDERED(THIS^.getTestNameFor('msbIsEqualTo')));

FOR multiplier := THIS^.FIRST_MULTIPLIER TO THIS^.LAST_MULTIPLIER DO
	valueToTest := ROR(THIS^.MULTIPLICAND * multiplier, THIS^.NUMBER_OF_RORS);

	THIS^.testMsbIsEqualTo(
		valueToTest := valueToTest,
		expectedValue := TRUE
	);	
	THIS^.testMsbIsEqualTo(
		valueToTest := valueToTest,
		expectedValue := FALSE
	);
END_FOR

THIS^.testMsbIsEqualTo(
	valueToTest := THIS^.LSB_ONLY,
	expectedValue := TRUE
);	
THIS^.testMsbIsEqualTo(
	valueToTest := THIS^.LSB_ONLY,
	expectedValue := FALSE
);
THIS^.testMsbIsEqualTo(
	valueToTest := THIS^.MSB_ONLY,
	expectedValue := TRUE
);	
THIS^.testMsbIsEqualTo(
	valueToTest := THIS^.MSB_ONLY,
	expectedValue := FALSE
);

TcUnit.TEST_FINISHED();
END_METHOD

(*

x summary
==================
This test method tests ``assert.bitNumber.x.msbIsNotEqualTo``
method of CNM_AssertionInterfaces library with various inputs

.. <legal notes>

legal notes
=================
| SPDX-FileCopyrightText: © 2022 ekvip automation GmbH <info@ekvip.de>
| SPDX-License-Identifier: Apache-2.0
| For details check: Apache-2.0_

.. _Apache-2.0: https://www.apache.org/licenses/LICENSE-2.0

.. </legal notes>

*)

METHOD runMsbIsNotEqualToTests
VAR
	(* it's just part of the test data *)
	valueToTest	:__XWORD;
	(* multiplier to get various bit patterns *)
	multiplier	:__UXINT;
END_VAR
RETURN (NOT TcUnit.TEST_ORDERED(THIS^.getTestNameFor('msbIsNotEqualTo')));

FOR multiplier := THIS^.FIRST_MULTIPLIER TO THIS^.LAST_MULTIPLIER DO
	valueToTest := ROR(THIS^.MULTIPLICAND * multiplier, THIS^.NUMBER_OF_RORS);
	THIS^.testMsbIsNotEqualTo(
		valueToTest := valueToTest,
		unexpectedValue := TRUE
	);	
	THIS^.testMsbIsNotEqualTo(
		valueToTest := valueToTest,
		unexpectedValue := FALSE
	);
END_FOR

THIS^.testMsbIsNotEqualTo(
	valueToTest := THIS^.LSB_ONLY,
	unexpectedValue := TRUE
);	
THIS^.testMsbIsNotEqualTo(
	valueToTest := THIS^.LSB_ONLY,
	unexpectedValue := FALSE
);
THIS^.testMsbIsNotEqualTo(
	valueToTest := THIS^.MSB_ONLY,
	unexpectedValue := TRUE
);	
THIS^.testMsbIsNotEqualTo(
	valueToTest := THIS^.MSB_ONLY,
	unexpectedValue := FALSE
);

TcUnit.TEST_FINISHED();
END_METHOD

(*

x summary
==================
This test method tests ``assert.bitNumber.x.msbIsSet``
of CNM_AssertionInterfaces library with various inputs

.. <legal notes>

legal notes
=================
| SPDX-FileCopyrightText: © 2022 ekvip automation GmbH <info@ekvip.de>
| SPDX-License-Identifier: Apache-2.0
| For details check: Apache-2.0_

.. _Apache-2.0: https://www.apache.org/licenses/LICENSE-2.0

.. </legal notes>

*)

METHOD runMsbIsSetTests
VAR
	(* it's just part of the test data *)
	valueToTest	:__XWORD;
	(* multiplier to get various bit patterns *)
	multiplier	:__UXINT;
END_VAR
RETURN (NOT TcUnit.TEST_ORDERED(THIS^.getTestNameFor('msbIsUnset')));

FOR multiplier := THIS^.FIRST_MULTIPLIER TO THIS^.LAST_MULTIPLIER DO
	valueToTest := ROR(THIS^.MULTIPLICAND * multiplier, THIS^.NUMBER_OF_RORS);
	THIS^.testMsbIsSet(
		valueToTest := valueToTest
	);
END_FOR

THIS^.testMsbIsSet(
	valueToTest := THIS^.LSB_ONLY
);	
THIS^.testMsbIsSet(
	valueToTest := THIS^.MSB_ONLY
);

TcUnit.TEST_FINISHED();
END_METHOD

(*

x summary
==================
This test method tests ``assert.bitNumber.x.msbIsUnset``
of CNM_AssertionInterfaces library with various inputs

.. <legal notes>

legal notes
=================
| SPDX-FileCopyrightText: © 2022 ekvip automation GmbH <info@ekvip.de>
| SPDX-License-Identifier: Apache-2.0
| For details check: Apache-2.0_

.. _Apache-2.0: https://www.apache.org/licenses/LICENSE-2.0

.. </legal notes>

*)

METHOD runMsbIsUnsetTests
VAR
	(* it's just part of the test data *)
	valueToTest	:__XWORD;
	(* multiplier to get various bit patterns *)
	multiplier	:__UXINT;
END_VAR
RETURN (NOT TcUnit.TEST_ORDERED(THIS^.getTestNameFor('msbIsSet')));

FOR multiplier := THIS^.FIRST_MULTIPLIER TO THIS^.LAST_MULTIPLIER DO
	valueToTest := ROR(THIS^.MULTIPLICAND * multiplier, THIS^.NUMBER_OF_RORS);
	THIS^.testMsbIsSet(
		valueToTest := valueToTest
	);
END_FOR

THIS^.testMsbIsSet(
	valueToTest := THIS^.LSB_ONLY
);	
THIS^.testMsbIsSet(
	valueToTest := THIS^.MSB_ONLY
);

TcUnit.TEST_FINISHED();
END_METHOD

(*

x summary
==================
This test method tests ``assert.bitNumber.x.orMaskIsEqualTo``
method of CNM_AssertionInterfaces library with various inputs

.. <legal notes>

legal notes
=================
| SPDX-FileCopyrightText: © 2022 ekvip automation GmbH <info@ekvip.de>
| SPDX-License-Identifier: Apache-2.0
| For details check: Apache-2.0_

.. _Apache-2.0: https://www.apache.org/licenses/LICENSE-2.0

.. </legal notes>

*)

METHOD runOrMaskIsEqualToTests
VAR
	(* shift to iterate through the bit numbers *)
	shift				:__UXINT;
	(* it's just part of the test data *)
	valueToTest		:__XWORD;
	(* mask with the bit iteration *)
	mask				:__XWORD;
END_VAR
RETURN (NOT TcUnit.TEST_ORDERED(THIS^.getTestNameFor('orMaskIsEqualTo')));

FOR shift:= THIS^.FIRST_BIT TO THIS^.LAST_BIT DO
	mask := SHL(THIS^.LSB_ONLY, shift);
	valueToTest := SHR(THIS^.MSB_ONLY, shift);
	THIS^.testOrMaskIsEqualTo(
		valueToTest := valueToTest,
		mask  := mask,
		expected := (mask OR valueToTest)
	);
	THIS^.testOrMaskIsEqualTo(
		valueToTest := valueToTest,
		mask  := mask,
		expected := (NOT (mask OR valueToTest))
	);
	THIS^.testAndMaskIsEqualTo(
		valueToTest := mask,
		mask  := (NOT mask),
		expected := THIS^.NO_BIT_SET
	);
	THIS^.testAndMaskIsEqualTo(
		valueToTest := mask,
		mask  := (NOT mask),
		expected := THIS^.ALL_BITS_SET
	);	
END_FOR

THIS^.testAndMaskIsEqualTo(
	valueToTest := THIS^.NO_BIT_SET,
	mask  := THIS^.NO_BIT_SET,
	expected := THIS^.NO_BIT_SET
);
THIS^.testAndMaskIsEqualTo(
	valueToTest := THIS^.NO_BIT_SET,
	mask  := THIS^.NO_BIT_SET,
	expected := THIS^.ALL_BITS_SET
);	

THIS^.testAndMaskIsEqualTo(
	valueToTest := THIS^.ALL_BITS_SET,
	mask  := THIS^.ALL_BITS_SET,
	expected := THIS^.ALL_BITS_SET
);
THIS^.testAndMaskIsEqualTo(
	valueToTest := THIS^.ALL_BITS_SET,
	mask  := THIS^.ALL_BITS_SET,
	expected := THIS^.NO_BIT_SET
);	

TcUnit.TEST_FINISHED();
END_METHOD

(*

x summary
==================
This test method tests ``assert.bitNumber.x.orMaskIsNotEqualTo``
method of CNM_AssertionInterfaces library with various inputs

.. <legal notes>

legal notes
=================
| SPDX-FileCopyrightText: © 2022 ekvip automation GmbH <info@ekvip.de>
| SPDX-License-Identifier: Apache-2.0
| For details check: Apache-2.0_

.. _Apache-2.0: https://www.apache.org/licenses/LICENSE-2.0

.. </legal notes>

*)

METHOD runOrMaskIsNotEqualToTests
VAR
	(* shift to iterate through the bit numbers *)
	shift				:__UXINT;
	(* it's just part of the test data *)
	valueToTest		:__XWORD;
	(* mask with the bit iteration *)
	mask				:__XWORD;
END_VAR
RETURN (NOT TcUnit.TEST_ORDERED(THIS^.getTestNameFor('orMaskIsNotEqualTo')));

FOR shift:= THIS^.FIRST_BIT TO THIS^.LAST_BIT DO
	mask := SHL(THIS^.LSB_ONLY, shift);
	valueToTest := SHR(THIS^.MSB_ONLY, shift);
	THIS^.testOrMaskIsNotEqualTo(
		valueToTest := valueToTest,
		mask  := mask,
		unexpected := (mask OR valueToTest)
	);
	THIS^.testOrMaskIsNotEqualTo(
		valueToTest := valueToTest,
		mask  := mask,
		unexpected := (NOT (mask OR valueToTest))
	);
	THIS^.testOrMaskIsNotEqualTo(
		valueToTest := mask,
		mask  := (NOT mask),
		unexpected := THIS^.NO_BIT_SET
	);
	THIS^.testOrMaskIsNotEqualTo(
		valueToTest := mask,
		mask  := (NOT mask),
		unexpected := THIS^.ALL_BITS_SET
	);	
END_FOR

THIS^.testOrMaskIsNotEqualTo(
	valueToTest := THIS^.NO_BIT_SET,
	mask  := THIS^.NO_BIT_SET,
	unexpected := THIS^.NO_BIT_SET
);
THIS^.testOrMaskIsNotEqualTo(
	valueToTest := THIS^.NO_BIT_SET,
	mask  := THIS^.NO_BIT_SET,
	unexpected := THIS^.ALL_BITS_SET
);	

THIS^.testOrMaskIsNotEqualTo(
	valueToTest := THIS^.ALL_BITS_SET,
	mask  := THIS^.ALL_BITS_SET,
	unexpected := THIS^.ALL_BITS_SET
);
THIS^.testOrMaskIsNotEqualTo(
	valueToTest := THIS^.ALL_BITS_SET,
	mask  := THIS^.ALL_BITS_SET,
	unexpected := THIS^.NO_BIT_SET
);	

TcUnit.TEST_FINISHED();
END_METHOD

(*

x summary
==================
This test method tests ``assert.bitNumber.x.valueIsEqualTo``
method of CNM_AssertionInterfaces library with various inputs

.. <legal notes>

legal notes
=================
| SPDX-FileCopyrightText: © 2022 ekvip automation GmbH <info@ekvip.de>
| SPDX-License-Identifier: Apache-2.0
| For details check: Apache-2.0_

.. _Apache-2.0: https://www.apache.org/licenses/LICENSE-2.0

.. </legal notes>

*)

METHOD runValueIsEqualToTests
RETURN (NOT TcUnit.TEST_ORDERED(THIS^.getTestNameFor('valueIsEqualTo')));

THIS^.testValueIsEqualTo(
	valueToTest := THIS^.NO_BIT_SET,
	expected := THIS^.ALL_BITS_SET
);
THIS^.testValueIsEqualTo(
	valueToTest := THIS^.NO_BIT_SET,
	expected := THIS^.NO_BIT_SET
);
THIS^.testValueIsEqualTo(
	valueToTest := THIS^.ALL_BITS_SET,
	expected := THIS^.ALL_BITS_SET
);
THIS^.testValueIsEqualTo(
	valueToTest := THIS^.ALL_BITS_SET,
	expected := THIS^.NO_BIT_SET
);
THIS^.testValueIsEqualTo(
	valueToTest := THIS^.LSB_ONLY,
	expected := THIS^.LSB_ONLY
);
THIS^.testValueIsEqualTo(
	valueToTest := THIS^.LSB_ONLY,
	expected := THIS^.MSB_ONLY
);
THIS^.testValueIsEqualTo(
	valueToTest := THIS^.MSB_ONLY,
	expected := THIS^.MSB_ONLY
);
THIS^.testValueIsEqualTo(
	valueToTest := THIS^.MSB_ONLY,
	expected := THIS^.LSB_ONLY
);

TcUnit.TEST_FINISHED();
END_METHOD

(*

x summary
==================
This test method tests ``assert.bitNumber.x.valueIsGreaterThan``
method of CNM_AssertionInterfaces library with various inputs

.. <legal notes>

legal notes
=================
| SPDX-FileCopyrightText: © 2022 ekvip automation GmbH <info@ekvip.de>
| SPDX-License-Identifier: Apache-2.0
| For details check: Apache-2.0_

.. _Apache-2.0: https://www.apache.org/licenses/LICENSE-2.0

.. </legal notes>

*)

METHOD runValueIsGreaterTests
RETURN (NOT TcUnit.TEST_ORDERED(THIS^.getTestNameFor('valueIsGreaterThan')));

THIS^.testValueIsGreater(
	valueToTest := THIS^.NO_BIT_SET,
	less := THIS^.ALL_BITS_SET
);
THIS^.testValueIsGreater(
	valueToTest := THIS^.NO_BIT_SET,
	less := THIS^.NO_BIT_SET
);
THIS^.testValueIsGreater(
	valueToTest := THIS^.ALL_BITS_SET,
	less := THIS^.ALL_BITS_SET
);
THIS^.testValueIsGreater(
	valueToTest := THIS^.ALL_BITS_SET,
	less := THIS^.NO_BIT_SET
);
THIS^.testValueIsGreater(
	valueToTest := THIS^.LSB_ONLY,
	less := THIS^.LSB_ONLY
);
THIS^.testValueIsGreater(
	valueToTest := THIS^.LSB_ONLY,
	less := THIS^.NO_BIT_SET
);
THIS^.testValueIsGreater(
	valueToTest := THIS^.LSB_ONLY,
	less := (THIS^.LSB_ONLY+THIS^.LSB_ONLY)
);
THIS^.testValueIsGreater(
	valueToTest := THIS^.MSB_ONLY,
	less := THIS^.MSB_ONLY
);
THIS^.testValueIsGreater(
	valueToTest := THIS^.MSB_ONLY,
	less := (NOT THIS^.MSB_ONLY)
);
THIS^.testValueIsGreater(
	valueToTest := THIS^.MSB_ONLY,
	less := THIS^.ALL_BITS_SET
);

TcUnit.TEST_FINISHED();
END_METHOD

(*

x summary
==================
This test method tests ``assert.bitNumber.x.valueIsInRangeOf``
method of CNM_AssertionInterfaces library with various inputs

.. <legal notes>

legal notes
=================
| SPDX-FileCopyrightText: © 2022 ekvip automation GmbH <info@ekvip.de>
| SPDX-License-Identifier: Apache-2.0
| For details check: Apache-2.0_

.. _Apache-2.0: https://www.apache.org/licenses/LICENSE-2.0

.. </legal notes>

*)

METHOD runValueIsInRangeOfTests
RETURN (NOT TcUnit.TEST_ORDERED(THIS^.getTestNameFor('valueIsInRangeOf')));

THIS^.testValueIsInRangeOf(
	lower := THIS^.NO_BIT_SET,
	valueToTest := THIS^.LSB_ONLY,
	upper := THIS^.ALL_BITS_SET
);
THIS^.testValueIsInRangeOf(
	lower := THIS^.NO_BIT_SET,
	valueToTest := THIS^.NO_BIT_SET,
	upper := THIS^.NO_BIT_SET
);
THIS^.testValueIsInRangeOf(
	lower := THIS^.ALL_BITS_SET,
	valueToTest := THIS^.ALL_BITS_SET,
	upper := THIS^.ALL_BITS_SET
);
THIS^.testValueIsInRangeOf(
	lower := THIS^.ALL_BITS_SET,
	valueToTest := THIS^.LSB_ONLY,
	upper := THIS^.NO_BIT_SET
);
THIS^.testValueIsInRangeOf(
	lower := THIS^.ALL_BITS_SET,
	valueToTest := THIS^.NO_BIT_SET,
	upper := THIS^.NO_BIT_SET
);

TEST_FINISHED();
END_METHOD

(*

x summary
==================
This test method tests ``assert.bitNumber.x.valueIsLessThan``
method of CNM_AssertionInterfaces library with various inputs

.. <legal notes>

legal notes
=================
| SPDX-FileCopyrightText: © 2022 ekvip automation GmbH <info@ekvip.de>
| SPDX-License-Identifier: Apache-2.0
| For details check: Apache-2.0_

.. _Apache-2.0: https://www.apache.org/licenses/LICENSE-2.0

.. </legal notes>

*)

METHOD runValueIsLessThanTests
RETURN (NOT TcUnit.TEST_ORDERED(THIS^.getTestNameFor('valueIsLessThan')));

THIS^.testValueIsLessThan(
	valueToTest := THIS^.NO_BIT_SET,
	greater := THIS^.ALL_BITS_SET
);
THIS^.testValueIsLessThan(
	valueToTest := THIS^.NO_BIT_SET,
	greater := THIS^.NO_BIT_SET
);
THIS^.testValueIsLessThan(
	valueToTest := THIS^.ALL_BITS_SET,
	greater := THIS^.ALL_BITS_SET
);
THIS^.testValueIsLessThan(
	valueToTest := THIS^.ALL_BITS_SET,
	greater := THIS^.NO_BIT_SET
);
THIS^.testValueIsLessThan(
	valueToTest := THIS^.LSB_ONLY,
	greater := THIS^.LSB_ONLY
);
THIS^.testValueIsLessThan(
	valueToTest := THIS^.LSB_ONLY,
	greater := THIS^.NO_BIT_SET
);
THIS^.testValueIsLessThan(
	valueToTest := THIS^.MSB_ONLY,
	greater := (THIS^.MSB_ONLY+THIS^.LSB_ONLY)
);
THIS^.testValueIsLessThan(
	valueToTest := THIS^.MSB_ONLY,
	greater := THIS^.MSB_ONLY
);
THIS^.testValueIsLessThan(
	valueToTest := THIS^.MSB_ONLY,
	greater := (NOT THIS^.MSB_ONLY)
);
THIS^.testValueIsLessThan(
	valueToTest := THIS^.MSB_ONLY,
	greater := THIS^.ALL_BITS_SET
);

TcUnit.TEST_FINISHED();
END_METHOD

(*

x summary
==================
This test method tests ``assert.bitNumber.x.valueIsMax``
method of CNM_AssertionInterfaces library with various inputs

.. <legal notes>

legal notes
=================
| SPDX-FileCopyrightText: © 2022 ekvip automation GmbH <info@ekvip.de>
| SPDX-License-Identifier: Apache-2.0
| For details check: Apache-2.0_

.. _Apache-2.0: https://www.apache.org/licenses/LICENSE-2.0

.. </legal notes>

*)

METHOD runValueIsMaxTests
RETURN (NOT TcUnit.TEST_ORDERED(THIS^.getTestNameFor('valueIsMax')));

THIS^.testValueIsMax(
	valueToTest := THIS^.NO_BIT_SET,
	maximum := THIS^.LSB_ONLY
);
THIS^.testValueIsMax(
	valueToTest := THIS^.LSB_ONLY,
	maximum := THIS^.NO_BIT_SET
);
THIS^.testValueIsMax(
	valueToTest := THIS^.NO_BIT_SET,
	maximum := THIS^.NO_BIT_SET
);
THIS^.testValueIsMax(
	valueToTest := THIS^.ALL_BITS_SET,
	maximum := ALL_BITS_SET
);
THIS^.testValueIsMax(
	valueToTest := (THIS^.ALL_BITS_SET-THIS^.LSB_ONLY),
	maximum := THIS^.ALL_BITS_SET
);
THIS^.testValueIsMax(
	valueToTest := THIS^.ALL_BITS_SET,
	maximum := (THIS^.ALL_BITS_SET-THIS^.LSB_ONLY)
);
THIS^.testValueIsMax(
	valueToTest := THIS^.MSB_ONLY,
	maximum := (THIS^.MSB_ONLY+THIS^.LSB_ONLY)
);
THIS^.testValueIsMax(
	valueToTest := (THIS^.MSB_ONLY+THIS^.LSB_ONLY),
	maximum := THIS^.MSB_ONLY
);
THIS^.testValueIsMax(
	valueToTest := THIS^.MSB_ONLY,
	maximum := (NOT THIS^.MSB_ONLY)
);
THIS^.testValueIsMax(
	valueToTest := (NOT THIS^.MSB_ONLY),
	maximum := THIS^.MSB_ONLY
);
THIS^.testValueIsMax(
	valueToTest := THIS^.MSB_ONLY,
	maximum := THIS^.MSB_ONLY
);

TcUnit.TEST_FINISHED();
END_METHOD

(*

x summary
==================
This test method tests ``assert.bitNumber.x.valueIsMin``
method of CNM_AssertionInterfaces library with various inputs

.. <legal notes>

legal notes
=================
| SPDX-FileCopyrightText: © 2022 ekvip automation GmbH <info@ekvip.de>
| SPDX-License-Identifier: Apache-2.0
| For details check: Apache-2.0_

.. _Apache-2.0: https://www.apache.org/licenses/LICENSE-2.0

.. </legal notes>

*)

METHOD runValueIsMinTests
RETURN (NOT TcUnit.TEST_ORDERED(THIS^.getTestNameFor('valueIsMin')));

THIS^.testValueIsMin(
	valueToTest := THIS^.NO_BIT_SET,
	minimum := THIS^.LSB_ONLY
);
THIS^.testValueIsMin(
	valueToTest := THIS^.LSB_ONLY,
	minimum := THIS^.NO_BIT_SET
);
THIS^.testValueIsMin(
	valueToTest := THIS^.NO_BIT_SET,
	minimum := THIS^.NO_BIT_SET
);
THIS^.testValueIsMin(
	valueToTest := THIS^.ALL_BITS_SET,
	minimum := ALL_BITS_SET
);
THIS^.testValueIsMin(
	valueToTest := (THIS^.ALL_BITS_SET-THIS^.LSB_ONLY),
	minimum := THIS^.ALL_BITS_SET
);
THIS^.testValueIsMin(
	valueToTest := THIS^.ALL_BITS_SET,
	minimum := (THIS^.ALL_BITS_SET-THIS^.LSB_ONLY)
);
THIS^.testValueIsMin(
	valueToTest := THIS^.MSB_ONLY,
	minimum := (THIS^.MSB_ONLY+THIS^.LSB_ONLY)
);
THIS^.testValueIsMin(
	valueToTest := (THIS^.MSB_ONLY+THIS^.LSB_ONLY),
	minimum := THIS^.MSB_ONLY
);
THIS^.testValueIsMin(
	valueToTest := THIS^.MSB_ONLY,
	minimum := (NOT THIS^.MSB_ONLY)
);
THIS^.testValueIsMin(
	valueToTest := (NOT THIS^.MSB_ONLY),
	minimum := THIS^.MSB_ONLY
);
THIS^.testValueIsMin(
	valueToTest := THIS^.MSB_ONLY,
	minimum := THIS^.MSB_ONLY
);

TcUnit.TEST_FINISHED();
END_METHOD

(*

x summary
==================
This test method tests ``assert.bitNumber.x.valueIsNotEqualTo``
method of CNM_AssertionInterfaces library with various inputs

.. <legal notes>

legal notes
=================
| SPDX-FileCopyrightText: © 2022 ekvip automation GmbH <info@ekvip.de>
| SPDX-License-Identifier: Apache-2.0
| For details check: Apache-2.0_

.. _Apache-2.0: https://www.apache.org/licenses/LICENSE-2.0

.. </legal notes>

*)

METHOD runValueIsNotEqualToTests
RETURN (NOT TcUnit.TEST_ORDERED(THIS^.getTestNameFor('valueIsNotEqualTo')));

THIS^.testValueIsNotEqualTo(
	valueToTest := THIS^.NO_BIT_SET,
	unexpected := THIS^.ALL_BITS_SET
);
THIS^.testValueIsNotEqualTo(
	valueToTest := THIS^.NO_BIT_SET,
	unexpected := THIS^.NO_BIT_SET
);
THIS^.testValueIsNotEqualTo(
	valueToTest := THIS^.ALL_BITS_SET,
	unexpected := THIS^.ALL_BITS_SET
);
THIS^.testValueIsNotEqualTo(
	valueToTest := THIS^.ALL_BITS_SET,
	unexpected := THIS^.NO_BIT_SET
);
THIS^.testValueIsNotEqualTo(
	valueToTest := THIS^.LSB_ONLY,
	unexpected := THIS^.LSB_ONLY
);
THIS^.testValueIsNotEqualTo(
	valueToTest := THIS^.LSB_ONLY,
	unexpected := THIS^.MSB_ONLY
);
THIS^.testValueIsNotEqualTo(
	valueToTest := THIS^.MSB_ONLY,
	unexpected := THIS^.MSB_ONLY
);
THIS^.testValueIsNotEqualTo(
	valueToTest := THIS^.MSB_ONLY,
	unexpected := THIS^.LSB_ONLY
);

TcUnit.TEST_FINISHED();
END_METHOD

(*

x summary
==================
This test method tests ``assert.bitNumber.x.xorMaskIsEqualTo``
method of CNM_AssertionInterfaces library with various inputs

.. <legal notes>

legal notes
=================
| SPDX-FileCopyrightText: © 2022 ekvip automation GmbH <info@ekvip.de>
| SPDX-License-Identifier: Apache-2.0
| For details check: Apache-2.0_

.. _Apache-2.0: https://www.apache.org/licenses/LICENSE-2.0

.. </legal notes>

*)

METHOD runXorMaskIsEqualToTests
VAR
	(* shift to iterate through the bit numbers *)
	shift				:__UXINT;
	(* it's just part of the test data *)
	valueToTest		:__XWORD;
	(* mask with the bit iteration *)
	mask				:__XWORD;
END_VAR
RETURN (NOT TcUnit.TEST_ORDERED(THIS^.getTestNameFor('xorMaskIsEqualTo')));

FOR shift:= THIS^.FIRST_BIT TO THIS^.LAST_BIT DO
	mask := SHL(THIS^.LSB_ONLY, shift);
	valueToTest := (NOT mask);
	THIS^.testOrMaskIsEqualTo(
		valueToTest := valueToTest,
		mask  := mask,
		expected := THIS^.ALL_BITS_SET
	);
	THIS^.testOrMaskIsEqualTo(
		valueToTest := valueToTest,
		mask  := mask,
		expected := THIS^.NO_BIT_SET
	);
	THIS^.testAndMaskIsEqualTo(
		valueToTest := mask,
		mask  := mask,
		expected := THIS^.NO_BIT_SET
	);
	THIS^.testAndMaskIsEqualTo(
		valueToTest := mask,
		mask  := mask,
		expected := mask
	);	
END_FOR

THIS^.testAndMaskIsEqualTo(
	valueToTest := THIS^.NO_BIT_SET,
	mask  := THIS^.NO_BIT_SET,
	expected := THIS^.NO_BIT_SET
);
THIS^.testAndMaskIsEqualTo(
	valueToTest := THIS^.NO_BIT_SET,
	mask  := THIS^.NO_BIT_SET,
	expected := THIS^.ALL_BITS_SET
);	

THIS^.testAndMaskIsEqualTo(
	valueToTest := THIS^.ALL_BITS_SET,
	mask  := THIS^.ALL_BITS_SET,
	expected := THIS^.ALL_BITS_SET
);
THIS^.testAndMaskIsEqualTo(
	valueToTest := THIS^.ALL_BITS_SET,
	mask  := THIS^.ALL_BITS_SET,
	expected := THIS^.NO_BIT_SET
);	

TcUnit.TEST_FINISHED();
END_METHOD

(*

x summary
==================
This test method tests ``assert.bitNumber.x.xorMaskIsNotEqualTo``
method of CNM_AssertionInterfaces library with various inputs

.. <legal notes>

legal notes
=================
| SPDX-FileCopyrightText: © 2022 ekvip automation GmbH <info@ekvip.de>
| SPDX-License-Identifier: Apache-2.0
| For details check: Apache-2.0_

